(* IEC 61131-3 sources: volt/packages/volt-lsp-iec/test-corpus/lenze-mid/Device/Plc Logic/Application/Library Manager/SymbolicVarsBase, 107 files *)

(* ---- ADDRESSOFINTERFACEUNION.dut ---- *)
TYPE ADDRESSOFINTERFACEUNION :
UNION
	IITF : __SYSTEM.IQueryInterface;
	IBASETREENODE : IBaseTreeNode;
	PITF : POINTER TO BYTE;
END_UNION
END_TYPE

(* ---- BROWSEOPERATION.dut ---- *)
TYPE BROWSEOPERATION :
(
	FIND_CHILD := 0,
	BROWSE_DOWN,
	BROWSE_NEXT,
	BROWSE_UP
);
END_TYPE

(* ---- CALLGLUEFUNCTIONPARAMETERSET.dut ---- *)
TYPE CALLGLUEFUNCTIONPARAMETERSET :
STRUCT
	PARGUMENTBUFFER : POINTER TO BYTE;
	NARGUMENTBUFFERSIZE : __XWORD;
	ITYPEDESC : REFERENCE TO TypeDesc;
	PINSTANCE : POINTER TO BYTE;
	PINTERFACE : __SYSTEM.IQueryInterface;
	RESULT : RTS_IEC_RESULT;
END_STRUCT
END_TYPE

(* ---- DIRECTIOBITS16.dut ---- *)
TYPE DIRECTIOBITS16 :
STRUCT
	X0 : BIT;
	X1 : BIT;
	X2 : BIT;
	X3 : BIT;
	X4 : BIT;
	X5 : BIT;
	X6 : BIT;
	X7 : BIT;
	X8 : BIT;
	X9 : BIT;
	X10 : BIT;
	X11 : BIT;
	X12 : BIT;
	X13 : BIT;
	X14 : BIT;
	X15 : BIT;
END_STRUCT
END_TYPE

(* ---- DIRECTIOBITS8.dut ---- *)
TYPE DIRECTIOBITS8 :
STRUCT
	X0 : BIT;
	X1 : BIT;
	X2 : BIT;
	X3 : BIT;
	X4 : BIT;
	X5 : BIT;
	X6 : BIT;
	X7 : BIT;
END_STRUCT
END_TYPE

(* ---- GETTYPENODEOPTIONS.dut ---- *)
TYPE GETTYPENODEOPTIONS :
(
	NOOPTION := 0,
	GETBASETYPE := 16#1,
	GETBROWSETYPE := 16#2
);
END_TYPE

(* ---- IECOPCUAMAPPING.dut ---- *)
TYPE IECOPCUAMAPPING :
STRUCT
	IECTYPE : TypeClass;
	UATYPE : OpcUa_BuiltInType;
	CONVERSIONNEEDED : BOOL;
END_STRUCT
END_TYPE

(* ---- LOGGERSTRING.dut ---- *)
TYPE LOGGERSTRING : STRING(255);
END_TYPE

(* ---- NESTINGPATHENTRY.dut ---- *)
TYPE NESTINGPATHENTRY :
STRUCT
	PPROPERTYINFO : POINTER TO PropertyInfo;
	PREFERENCEINFO : POINTER TO BYTE;
	CONTAININGNODE : ILeafTreeNode;
	NNEXTOFFSET : __XWORD;
	PTYPENODE : REFERENCE TO TypeDesc;
END_STRUCT
END_TYPE

(* ---- NESTINGPATHINFORMATION.dut ---- *)
TYPE NESTINGPATHINFORMATION :
STRUCT
	NMAXDEPTH : UDINT;
	NELEMENTSUSED : UDINT;
	APATHINFO : ARRAY [0..5] OF NestingPathEntry;
END_STRUCT
END_TYPE

(* ---- NODEFLAGS.dut ---- *)
TYPE NODEFLAGS :
(
	LTNF_NONE := 16#0,
	LTNF_VAR := 16#1,
	LTNF_VAR_INPUT := 16#2,
	LTNF_VAR_OUTPUT := 16#4,
	LTNF_VAR_IN_OUT := 16#8,
	LTNF_VAR_EXEC := 16#10,
	LTNF_VAR_PROP := 16#20,
	LTNF_CALL_PROP := 16#40,
	LTNF_INHERITED_MEMBER := 16#10000
);
END_TYPE

(* ---- OPCUAMETADATATYPE.dut ---- *)
TYPE OPCUAMETADATATYPE :
(
	WELLKNOWNDATATYPEMETA := 0,
	OWNDATATYPEMETA,
	METHODMETA
);
END_TYPE

(* ---- OPCUAMETHODMETADATA.dut ---- *)
TYPE OPCUAMETHODMETADATA :
STRUCT
	INPUTARGUMENTS : OpcUa_NodeId;
	OUTPUTARGUMENTS : OpcUa_NodeId;
END_STRUCT
END_TYPE

(* ---- OPCUANODEMETADATA.dut ---- *)
TYPE OPCUANODEMETADATA :
STRUCT
	BROWSENAME : OpcUa_QualifiedName;
	DISPLAYNAME : OpcUa_LocalizedText;
	NODECLASS : OpcUa_NodeClass;
	DESCRIPTION : OpcUa_LocalizedText;
	EVENTNOTIFIER : OpcUa_Byte;
	REFERENCEPARENT : OpcUa_NodeId;
	TYPEDEFINITION : OpcUa_NodeId;
	ENTRYPOINT : OpcUa_NodeId;
END_STRUCT
END_TYPE

(* ---- OPCUAOWNDATATYPEMETADATA.dut ---- *)
TYPE OPCUAOWNDATATYPEMETADATA :
STRUCT
	PARENTID : OpcUa_NodeId;
	PARTENTREFERENCETYPE : OpcUa_NodeId;
END_STRUCT
END_TYPE

(* ---- OPCUATYPEMETADATA.dut ---- *)
TYPE OPCUATYPEMETADATA :
STRUCT
	METATYPE : OpcUaMetaDataType;
	DATA : OpcUaTypeMetaDataUnion;
END_STRUCT
END_TYPE

(* ---- OPCUATYPEMETADATAUNION.dut ---- *)
TYPE OPCUATYPEMETADATAUNION :
UNION
	WELLKNOWN : OpcUaWellKnownDataTypeMetaData;
	OWNDATATYPE : OpcUaOwnDataTypeMetaData;
	METHODDATA : OpcUaMethodMetaData;
END_UNION
END_TYPE

(* ---- OPCUAWELLKNOWNDATATYPEMETADATA.dut ---- *)
TYPE OPCUAWELLKNOWNDATATYPEMETADATA :
STRUCT
	NODEID : OpcUa_NodeId;
	ENCODINGID : OpcUa_NodeId;
END_STRUCT
END_TYPE

(* ---- PROPERTYINFO.dut ---- *)
TYPE PROPERTYINFO :
STRUCT
	PINSTANCE : POINTER TO BYTE;
	PPFGET : POINTER TO POINTER TO BYTE;
	PPFSET : POINTER TO POINTER TO BYTE;
	_NPROPOFFSETGET : INT;
	_NPROPOFFSETSET : INT;
END_STRUCT
END_TYPE

(* ---- PROPERTYINFOREMOTE.dut ---- *)
TYPE PROPERTYINFOREMOTE :
STRUCT
	AREACODE : INT;
	OFFSETGET : DINT;
	OFFSETSET : DINT;
END_STRUCT
END_TYPE

(* ---- SYMBOLICVARSBASEHANDLECONVERTER.dut ---- *)
TYPE SYMBOLICVARSBASEHANDLECONVERTER :
UNION
	HHANDLE : RTS_IEC_HANDLE;
	PBASENODE : IBaseTreeNode;
	PTYPEDESC : ITypeDesc;
END_UNION
END_TYPE

(* ---- GVL_LIBRARYDEFINES.gvl ---- *)
VAR_GLOBAL
	IECVARACCESS_VERSION_GE_3_1_3_0 : INT := 1;
	IECVARACCESS_VERSION_GE_3_2_0_1 : INT := 2;
	CMPID_IECVARACCESS : DWORD := 16#1007;
	IECVARACCESS_LIB_VERSION : DWORD := 16#3050340;
	CMPNAME_IECVARACCESS : STRING := 'IecVarAccess';
END_VAR

(* ---- IECUAMAPPING.gvl ---- *)
VAR_GLOBAL
	MAPPING : ARRAY [0..49] OF IecOpcUaMapping := [STRUCT(iecType := TYPE_BOOL, uaType := OpcUaType_Boolean), STRUCT(iecType := TYPE_BIT, uaType := OpcUaType_Boolean), STRUCT(iecType := TYPE_BYTE, uaType := OpcUaType_Byte), STRUCT(iecType := TYPE_WORD, uaType := OpcUaType_UInt16), STRUCT(iecType := TYPE_DWORD, uaType := OpcUaType_UInt32), STRUCT(iecType := TYPE_LWORD, uaType := OpcUaType_UInt64), STRUCT(iecType := TYPE_SINT, uaType := OpcUaType_SByte), STRUCT(iecType := TYPE_INT, uaType := OpcUaType_Int16), STRUCT(iecType := TYPE_DINT, uaType := OpcUaType_Int32), STRUCT(iecType := TYPE_LINT, uaType := OpcUaType_Int64), STRUCT(iecType := TYPE_USINT, uaType := OpcUaType_Byte), STRUCT(iecType := TYPE_UINT, uaType := OpcUaType_UInt16), STRUCT(iecType := TYPE_UDINT, uaType := OpcUaType_UInt32), STRUCT(iecType := TYPE_ULINT, uaType := OpcUaType_UInt64), STRUCT(iecType := TYPE_REAL, uaType := OpcUaType_Float), STRUCT(iecType := TYPE_LREAL, uaType := OpcUaType_Double), STRUCT(iecType := TYPE_STRING, uaType := OpcUaType_String), STRUCT(iecType := TYPE_WSTRING, uaType := OpcUaType_String), STRUCT(iecType := TYPE_TIME, uaType := OpcUaType_Int64), STRUCT(iecType := TYPE_DATE, uaType := OpcUaType_DateTime), STRUCT(iecType := TYPE_DATEANDTIME, uaType := OpcUaType_DateTime), STRUCT(iecType := TYPE_TIMEOFDAY, uaType := OpcUaType_UInt32), STRUCT(iecType := TYPE_POINTER, uaType := OpcUaType_Null), STRUCT(iecType := TYPE_REFERENCE, uaType := OpcUaType_Null), STRUCT(iecType := TYPE_SUBRANGE, uaType := OpcUaType_Null), STRUCT(iecType := TYPE_ENUM, uaType := OpcUaType_Null), STRUCT(iecType := TYPE_ARRAY, uaType := OpcUaType_Null), STRUCT(iecType := TYPE_PARAMS, uaType := OpcUaType_Null), STRUCT(iecType := TYPE_USERDEF, uaType := OpcUaType_ExtensionObject), STRUCT(iecType := TYPE_NONE, uaType := OpcUaType_Null), STRUCT(iecType := TYPE_ANY, uaType := OpcUaType_Null), STRUCT(iecType := TYPE_ANYBIT, uaType := OpcUaType_Null), STRUCT(iecType := TYPE_ANYDATE, uaType := OpcUaType_Null), STRUCT(iecType := TYPE_ANYINT, uaType := OpcUaType_Null), STRUCT(iecType := TYPE_ANYNUM, uaType := OpcUaType_Null), STRUCT(iecType := TYPE_ANYREAL, uaType := OpcUaType_Null), STRUCT(iecType := TYPE_LAZY, uaType := OpcUaType_Null), STRUCT(iecType := TYPE_LTIME, uaType := OpcUaType_Int64), STRUCT(iecType := TYPE_BITCONST, uaType := OpcUaType_Null), STRUCT(iecType := TYPE_UXINT, uaType := OpcUaType_Null), STRUCT(iecType := TYPE_XWORD, uaType := OpcUaType_Null), STRUCT(iecType := TYPE_XINT, uaType := OpcUaType_Null), STRUCT(iecType := TYPE_XSRTING, uaType := OpcUaType_Null), STRUCT(iecType := TYPE_VARLENARRAY, uaType := OpcUaType_Null), STRUCT(iecType := TYPE_ANYSTRING, uaType := OpcUaType_Null), STRUCT(iecType := TYPE_VECTOR, uaType := OpcUaType_Null), STRUCT(iecType := TYPE_LDATE, uaType := OpcUaType_Null), STRUCT(iecType := TYPE_LDATEANDTIME, uaType := OpcUaType_Null), STRUCT(iecType := TYPE_LTIMEOFDAY, uaType := OpcUaType_Null), STRUCT(iecType := TYPE_INTERFACE, uaType := OpcUaType_Null)];
	SECS_BETWEEN_EPOCHS : LINT := 11644473600;
	SECS_TO_100NS : LINT := 10000000;
END_VAR

(* ---- INTERFACEIDS.gvl ---- *)
VAR_GLOBAL
	ITFID_ICOLLECTSSECONDOFFSET : DWORD := 16#1003;
	ITFID_ICOLLECTSPROPERTYINFORMATION : DWORD := 16#1004;
	ITFID_ILEAFTREENODE : DWORD := 16#1006;
	ITFID_IBRANCHTREENODE : DWORD := 16#1011;
	ITFID_IMEMBERINDEX : DWORD := 16#1012;
	ITFID_IARRAYNOTIFIABLE : DWORD := 16#1030;
	ITFID_IVARIABLEINFORMATIONCOMBINED : DWORD := 16#1105;
	ITFID_ITREEWALKER : DWORD := 16#1111;
END_VAR

(* ---- POUTYPECLASS.gvl ---- *)
VAR_GLOBAL
	TYPE_POU_FUNCTION : INT := 16#100;
	TYPE_POU_FUNCTION_BLOCK : INT := 16#200;
	TYPE_POU_PROGRAM : INT := 16#300;
	TYPE_POU_STRUCTURE : INT := 16#400;
	TYPE_POU_UNION : INT := 16#500;
	TYPE_POU_UABUILTIN : INT := 16#1000;
END_VAR

(* ---- TYPECLASSFLAGBITS.gvl ---- *)
VAR_GLOBAL
	TYPECLASS_FLAG_ALIAS : INT := 16#900;
	TYPECLASS_MAGIC_PROPERTY : INT := ANY_TO_INT(16#E000);
	TYPECLASS_BITMASK_TYPECLASS : INT := 16#FF;
	TYPECLASS_BITMASK_POUTYPE : INT := 16#700;
	TYPECLASS_BITMASK_FLAGS : INT := ANY_TO_INT(16#F800);
END_VAR

(* ---- TYPEFLAGS.gvl ---- *)
VAR_GLOBAL
	TYPEFLAG_REFERENCE : DWORD := 16#1;
END_VAR

(* ---- IARRAYNOTIFIABLE.itf ---- *)
INTERFACE IARRAYNOTIFIABLE
END_INTERFACE

METHOD ARRAYACCESSDETECTED
VAR_INPUT
	PSTR : POINTER TO STRING;
	LENGTH : INT;
END_VAR
END_METHOD

(* ---- IBRANCHTREENODE.itf ---- *)
INTERFACE IBRANCHTREENODE
END_INTERFACE

METHOD GETATTRIBUTEBYINDEX : POINTER TO STRING
VAR_INPUT
	WINDEX : WORD;
END_VAR
END_METHOD

METHOD GETNAMESPACENODEFLAGS : IecVarAccess_Interfaces.NamespaceNodeFlags
VAR_INPUT
	PRESULT : POINTER TO UDINT;
END_VAR
END_METHOD

METHOD GETNUMOFATTRIBUTES : WORD
END_METHOD

(* ---- ILEAFTREENODE.itf ---- *)
INTERFACE ILEAFTREENODE
END_INTERFACE

METHOD EXECUTECALL : RTS_IEC_RESULT
VAR_INPUT
	VARINFO : REFERENCE TO VariableInformation;
	PARGUMENTBUFFER : POINTER TO BYTE;
	NARGUMENTBUFFERSIZE : __XWORD;
	CALLEXECUTORFUNCTION : POINTER TO POINTER TO BYTE;
	EXECUTABLETYPEDESC : REFERENCE TO TypeDesc;
END_VAR
END_METHOD

METHOD EXECUTECALL2 : RTS_IEC_RESULT
VAR_INPUT
	VARINFO : REFERENCE TO VariableInformation;
	PARGUMENTBUFFER : POINTER TO BYTE;
	NARGUMENTBUFFERSIZE : __XWORD;
END_VAR
END_METHOD

METHOD GET : __XWORD
VAR_INPUT
	PDEST : POINTER TO BYTE;
	VARINFO : REFERENCE TO VariableInformation;
	DWSIZE : __XWORD;
	PRESULT : POINTER TO RTS_IEC_RESULT;
END_VAR
END_METHOD

METHOD GETACCESSRIGHTS : BYTE
END_METHOD

METHOD GETACCESSRIGHTS2 : BYTE
VAR_INPUT
	VARINFO : REFERENCE TO VariableInformation;
	BGETUSERRIGHTS : BOOL;
END_VAR
END_METHOD

METHOD GETADDRESS : POINTER TO BYTE
END_METHOD

METHOD GETADDRESS3 : POINTER TO BYTE
VAR_INPUT
	PVARIABLEINFORMATION : POINTER TO VariableInformationStruct;
END_VAR
END_METHOD

METHOD GETATTRIBUTEBYINDEX : POINTER TO STRING
VAR_INPUT
	WINDEX : WORD;
END_VAR
END_METHOD

METHOD GETCLIENTOFFSET : DWORD
END_METHOD

METHOD GETFLAGS : NodeFlags
END_METHOD

METHOD GETNAMESPACENODEFLAGS : IecVarAccess_Interfaces.NamespaceNodeFlags
VAR_INPUT
	PRESULT : POINTER TO UDINT;
END_VAR
END_METHOD

METHOD GETNUMOFATTRIBUTES : WORD
END_METHOD

METHOD GETSIZE : __XWORD
VAR_INPUT
	VARINFO : REFERENCE TO VariableInformation;
	PRESULT : POINTER TO RTS_IEC_RESULT;
END_VAR
END_METHOD

METHOD GETTYPE : REFERENCE TO TypeDesc
VAR_INPUT
	VARINFO : REFERENCE TO VariableInformation;
	OPTIONS : WORD;
END_VAR
END_METHOD

METHOD NODEFOUND : UDINT
VAR_INPUT
	VARINFO : REFERENCE TO VariableInformation;
	BDIRECTCHILDFOUND : BOOL;
END_VAR
END_METHOD

METHOD SET : __XWORD
VAR_INPUT
	PSRC : POINTER TO BYTE;
	VARINFO : REFERENCE TO VariableInformation;
	DWSIZE : __XWORD;
	PRESULT : POINTER TO RTS_IEC_RESULT;
END_VAR
END_METHOD

METHOD SWAP2 : __XWORD
VAR_INPUT
	PDATA : POINTER TO BYTE;
	VARINFO : REFERENCE TO VariableInformation;
	BMOTOROLA : BOOL;
	PRESULT : POINTER TO RTS_IEC_RESULT;
END_VAR
END_METHOD

(* ---- IMEMBERINDEX.itf ---- *)
INTERFACE IMEMBERINDEX
END_INTERFACE

(* ---- IOPCUADATATYPEFINDCHILDBYBROWSENAME.itf ---- *)
INTERFACE IOPCUADATATYPEFINDCHILDBYBROWSENAME
END_INTERFACE

METHOD GETFIRSTCHILDBYBROWSENAME : ITreeWalker
VAR_INPUT
	PBROWSENAME : POINTER TO OpcUa_QualifiedName;
	VARINFO : REFERENCE TO VariableInformation;
END_VAR
VAR_OUTPUT
	RESULT : RTS_IEC_RESULT;
END_VAR
END_METHOD

(* ---- IOPCUADATATYPEMETADATA.itf ---- *)
INTERFACE IOPCUADATATYPEMETADATA
END_INTERFACE

METHOD GETDATATYPEID : RTS_IEC_RESULT
VAR_OUTPUT
	PDATATYPEID : POINTER TO OpcUa_NodeId;
END_VAR
END_METHOD

METHOD GETENCODINGNODEID : RTS_IEC_RESULT
VAR_OUTPUT
	PENCODINGID : POINTER TO OpcUa_NodeId;
END_VAR
END_METHOD

METHOD GETMETHODARGUMENTS : RTS_IEC_RESULT
VAR_OUTPUT
	PINPUTARGUMENTS : POINTER TO OpcUa_NodeId;
	POUTPUTARGUMENTS : POINTER TO OpcUa_NodeId;
END_VAR
END_METHOD

METHOD GETPARENTNODE : RTS_IEC_RESULT
VAR_OUTPUT
	PPARENTNODE : POINTER TO OpcUa_NodeId;
END_VAR
END_METHOD

METHOD GETPARENTREFERENCETYPE : RTS_IEC_RESULT
VAR_OUTPUT
	PPARENTREFERENCETYPE : POINTER TO OpcUa_NodeId;
END_VAR
END_METHOD

METHOD ISWELLKNOWNTYPE : BOOL
END_METHOD

(* ---- IOPCUAINSTANCEMETADATA.itf ---- *)
INTERFACE IOPCUAINSTANCEMETADATA
END_INTERFACE

METHOD GETBROWSENAME : RTS_IEC_RESULT
VAR_OUTPUT
	PBROWSENAME : POINTER TO OpcUa_QualifiedName;
END_VAR
END_METHOD

METHOD GETDESCRIPTION : RTS_IEC_RESULT
VAR_OUTPUT
	PDESCRIPTION : POINTER TO OpcUa_LocalizedText;
END_VAR
END_METHOD

METHOD GETDISPLAYNAME : RTS_IEC_RESULT
VAR_OUTPUT
	PDISPLAYNAME : POINTER TO OpcUa_LocalizedText;
END_VAR
END_METHOD

METHOD GETENTRYPOINT : RTS_IEC_RESULT
VAR_OUTPUT
	ISENTRYPOINT : BOOL;
	PENTRYPOINT : POINTER TO CmpOPCUAStack_Interfaces.OpcUa_NodeId;
END_VAR
END_METHOD

METHOD GETEVENTNOTIFIER : RTS_IEC_RESULT
VAR_OUTPUT
	EVENTNOTIFIER : OpcUa_Byte;
END_VAR
END_METHOD

METHOD GETNODECLASS : RTS_IEC_RESULT
VAR_OUTPUT
	NODECLASS : OpcUa_NodeClass;
END_VAR
END_METHOD

METHOD GETPARENTREFERENCETYPE : RTS_IEC_RESULT
VAR_OUTPUT
	PREFERENCETYPE : POINTER TO OpcUa_NodeId;
END_VAR
END_METHOD

METHOD GETTYPEDEFINITION : RTS_IEC_RESULT
VAR_OUTPUT
	PTYPEDEFINITION : POINTER TO OpcUa_NodeId;
END_VAR
END_METHOD

(* ---- ISEARCHCALLBACKS.itf ---- *)
INTERFACE ISEARCHCALLBACKS
END_INTERFACE

METHOD IGNOREROOTNODE : BOOL
VAR_INPUT
	PNODE : ITreeWalker;
	VARINFO : REFERENCE TO VariableInformation;
END_VAR
END_METHOD

METHOD NODEFOUND
VAR_INPUT
	PNODE : ITreeWalker;
	VARINFO : REFERENCE TO VariableInformation;
	XROOTNODE : BOOL;
END_VAR
END_METHOD

METHOD NODENOTFOUND : ITreeWalker
VAR_INPUT
	PPARENT : ITreeWalker;
	SZCHILDNAME : POINTER TO BYTE;
	NAMELEN : __XWORD;
	SYMBOLSSETS : DWORD;
	VARINFO : REFERENCE TO VariableInformation;
	XROOTNODE : BOOL;
END_VAR
VAR_IN_OUT
	CONSUMED : __XWORD;
END_VAR
END_METHOD

(* ---- ITREEWALKER.itf ---- *)
INTERFACE ITREEWALKER
END_INTERFACE

METHOD ASBASETREENODE : IBaseTreeNode
END_METHOD

METHOD FINDCHILD : ITreeWalker
VAR_INPUT
	SZCHILDNAME : POINTER TO BYTE;
	NAMELEN : __XWORD;
	SYMBOLSSETS : DWORD;
	VARINFO : REFERENCE TO VariableInformation;
	PRESULT : POINTER TO RTS_IEC_RESULT;
END_VAR
VAR_IN_OUT
	TYPESYSTEMREACHED : BOOL;
END_VAR
END_METHOD

METHOD GETCHILDBYINDEX : ITreeWalker
VAR_INPUT
	IINDEX : DINT;
	USERACCESSRIGHTS : BYTE;
	SYMBOLSSETS : DWORD;
END_VAR
VAR_OUTPUT
	XOUTOFRANGE : BOOL;
END_VAR
END_METHOD

METHOD GETFIRSTCHILD : ITreeWalker
VAR_INPUT
	USERACCESSRIGHTS : BYTE;
	SYMBOLSSETS : DWORD;
END_VAR
END_METHOD

METHOD GETFULLPATH : DINT
VAR_INPUT
	PBUFFER : POINTER TO STRING;
	DIBUFFERSIZE : DINT;
END_VAR
VAR_OUTPUT
	BROOT_NODE : BOOL;
	BEMPTYNAMESPACENODE : BOOL;
END_VAR
END_METHOD

METHOD GETPARENT : ITreeWalker
VAR_INPUT
	USERACCESSRIGHTS : BYTE;
	SYMBOLSSETS : DWORD;
END_VAR
END_METHOD

METHOD GETSIBLING : ITreeWalker
VAR_INPUT
	USERACCESSRIGHTS : BYTE;
	SYMBOLSSETS : DWORD;
END_VAR
END_METHOD

METHOD ISVISIBLE : BOOL
VAR_INPUT
	USERACCESSRIGHTS : BYTE;
	SYMBOLSSETS : DWORD;
END_VAR
END_METHOD

METHOD GETCHILDBYBROWSENAME : ITreeWalker
VAR_INPUT
	PBROWSENAME : POINTER TO OpcUa_QualifiedName;
	VARINFO : REFERENCE TO VariableInformation;
END_VAR
END_METHOD

METHOD GETNEXTBYBROWSENAME : ITreeWalker
VAR_INPUT
	PBROWSENAME : POINTER TO OpcUa_QualifiedName;
	VARINFO : REFERENCE TO VariableInformation;
END_VAR
END_METHOD

(* ---- ADDRESSOFIBASETREENODE.pou ---- *)
FUNCTION ADDRESSOFIBASETREENODE : POINTER TO BYTE
VAR_INPUT
	IBASETREENODE : IBaseTreeNode;
END_VAR
END_FUNCTION

(* ---- ADDRESSOFINTERFACE.pou ---- *)
FUNCTION ADDRESSOFINTERFACE : POINTER TO BYTE
VAR_INPUT
	IITF : __SYSTEM.IQueryInterface;
END_VAR
END_FUNCTION

(* ---- ASCIIUPPER.pou ---- *)
FUNCTION ASCIIUPPER : BYTE
VAR_INPUT
	CHARACTER : BYTE;
END_VAR
END_FUNCTION

(* ---- CALCULATEPROPERTYBUFFERSIZE.pou ---- *)
FUNCTION CALCULATEPROPERTYBUFFERSIZE : __XWORD
VAR_INPUT
	DATATYPE : REFERENCE TO TypeDesc;
END_VAR
END_FUNCTION

(* ---- CALLGLUEDESERIALIZEPARAMETERS.pou ---- *)
FUNCTION CALLGLUEDESERIALIZEPARAMETERS : RTS_IEC_RESULT
VAR_INPUT
	PARGUMENTBUFFER : POINTER TO BYTE;
	NARGUMENTBUFFERSIZE : __XWORD;
	ITYPEDESC : REFERENCE TO TypeDesc;
	PPARSEDARGUMENTS : POINTER TO BYTE;
	NPARSEDARGUMENTSIZE : __XWORD;
END_VAR
END_FUNCTION

(* ---- CALLGLUESERIALIZERETURNVALUES.pou ---- *)
FUNCTION CALLGLUESERIALIZERETURNVALUES : RTS_IEC_RESULT
VAR_INPUT
	PARGUMENTBUFFER : POINTER TO BYTE;
	NARGUMENTBUFFERSIZE : __XWORD;
	ITYPEDESC : REFERENCE TO TypeDesc;
	PPARSEDARGUMENTS : POINTER TO BYTE;
	NPARSEDARGUMENTSIZE : __XWORD;
END_VAR
END_FUNCTION

(* ---- COMPAREBROWSENAME.pou ---- *)
FUNCTION COMPAREBROWSENAME : DINT
VAR_INPUT
	NAME1 : POINTER TO OpcUa_QualifiedName;
	NAME2 : POINTER TO OpcUa_QualifiedName;
END_VAR
END_FUNCTION

(* ---- CONVERTTOIBRANCHTREENODE.pou ---- *)
FUNCTION CONVERTTOIBRANCHTREENODE : IBranchTreeNode
VAR_INPUT
	PNODE : IBaseTreeNode;
END_VAR
END_FUNCTION

(* ---- CONVERTTOILEAFTREENODE.pou ---- *)
FUNCTION CONVERTTOILEAFTREENODE : ILeafTreeNode
VAR_INPUT
	PNODE : IBaseTreeNode;
END_VAR
END_FUNCTION

(* ---- CONVERTTOITREEWALKER.pou ---- *)
FUNCTION CONVERTTOITREEWALKER : ITreeWalker
VAR_INPUT
	PNODE : IBaseTreeNode;
END_VAR
END_FUNCTION

(* ---- FINDBYBROWSENAME.pou ---- *)
FUNCTION FINDBYBROWSENAME : POINTER TO SymbolsBaseNode
VAR_INPUT
	LIST : POINTER TO POINTER TO SymbolsBaseNode;
	NUMELEMENTS : DINT;
	PBROWSENAME : POINTER TO OpcUa_QualifiedName;
END_VAR
VAR_OUTPUT
	INDEX : DINT;
END_VAR
END_FUNCTION

(* ---- FINDNEXTBYBROWSENAME.pou ---- *)
FUNCTION FINDNEXTBYBROWSENAME : POINTER TO SymbolsBaseNode
VAR_INPUT
	LIST : POINTER TO POINTER TO SymbolsBaseNode;
	NUMELEMENTS : DINT;
	PBROWSENAME : POINTER TO OpcUa_QualifiedName;
	VARINFO : REFERENCE TO VariableInformation;
END_VAR
VAR_OUTPUT
	RESULT : RTS_IEC_RESULT;
END_VAR
VAR_IN_OUT
	INDEX : DINT;
END_VAR
END_FUNCTION

(* ---- HEXSTRING.pou ---- *)
FUNCTION HEXSTRING : STRING
VAR_INPUT
	UDIVALUE : __UXINT;
END_VAR
END_FUNCTION

(* ---- ISACCEPTEDLEAFNODE.pou ---- *)
FUNCTION ISACCEPTEDLEAFNODE : BOOL
VAR_INPUT
	NITYPE : INT;
END_VAR
END_FUNCTION

(* ---- ISINVALIDMEMORYADDRESS.pou ---- *)
FUNCTION ISINVALIDMEMORYADDRESS : BOOL
VAR_INPUT
	PDATA : POINTER TO BYTE;
	XWSIZE : __XWORD;
	BWRITE : BOOL;
	PRESULT : POINTER TO RTS_IEC_RESULT;
END_VAR
END_FUNCTION

(* ---- ITREEWALKER_TOSTRING.pou ---- *)
FUNCTION ITREEWALKER_TOSTRING : LoggerString
VAR_INPUT
	ITREEWALKER : ITreeWalker;
END_VAR
END_FUNCTION

(* ---- LEAFTREENODE_TOSTRING.pou ---- *)
FUNCTION LEAFTREENODE_TOSTRING : LoggerString
VAR_INPUT
	LEAFTREENODE : POINTER TO LeafTreeNode;
END_VAR
END_FUNCTION

(* ---- LOGERROR.pou ---- *)
FUNCTION LOGERROR
VAR_INPUT
	STR : LoggerString;
END_VAR
END_FUNCTION

(* ---- LOGINFO.pou ---- *)
FUNCTION LOGINFO
VAR_INPUT
	STR : LoggerString;
END_VAR
END_FUNCTION

(* ---- LOGSTRING.pou ---- *)
FUNCTION LOGSTRING
VAR_INPUT
	STR : LoggerString;
	LOGCLASS : UDINT := CmpLog.LogClass.LOG_INFO;
END_VAR
END_FUNCTION

(* ---- MEMCPY.pou ---- *)
FUNCTION MEMCPY : __XWORD
VAR_INPUT
	PBYDEST : POINTER TO BYTE;
	PBYSRC : POINTER TO BYTE;
	DWSIZE : __XWORD;
END_VAR
END_FUNCTION

(* ---- MEMSET.pou ---- *)
FUNCTION MEMSET : __XWORD
VAR_INPUT
	PBYDEST : POINTER TO BYTE;
	BYVALUE : BYTE;
	DWSIZE : __XWORD;
END_VAR
END_FUNCTION

(* ---- PSTRCAT.pou ---- *)
FUNCTION PSTRCAT : DINT
VAR_INPUT
	PSTDEST : POINTER TO STRING;
	PSTSRC : POINTER TO STRING;
	DIDESTSIZE : DINT;
END_VAR
END_FUNCTION

(* ---- PSTRCMP.pou ---- *)
FUNCTION PSTRCMP : INT
VAR_INPUT
	PSTR1 : POINTER TO STRING;
	PSTR2 : POINTER TO STRING;
END_VAR
END_FUNCTION

(* ---- PSTRICMP.pou ---- *)
FUNCTION PSTRICMP : INT
VAR_INPUT
	PSTR1 : POINTER TO STRING;
	PSTR2 : POINTER TO STRING;
END_VAR
END_FUNCTION

(* ---- PSTRLEN.pou ---- *)
FUNCTION PSTRLEN : DINT
VAR_INPUT
	PSTRING : POINTER TO STRING;
END_VAR
END_FUNCTION

(* ---- PSTRLENUNTIL.pou ---- *)
FUNCTION PSTRLENUNTIL : DINT
VAR_INPUT
	PST : POINTER TO STRING;
	STTOKENDELIMITERS : STRING;
END_VAR
END_FUNCTION

(* ---- PSTRNICMP.pou ---- *)
FUNCTION PSTRNICMP : INT
VAR_INPUT
	PSTR1 : POINTER TO STRING;
	PSTR2 : POINTER TO STRING;
	N : __XWORD;
END_VAR
END_FUNCTION

(* ---- REPARSEIOMEMORYACCESSEXPRESSION.pou ---- *)
FUNCTION REPARSEIOMEMORYACCESSEXPRESSION : BOOL
VAR_INPUT
	STDESTINATION : REFERENCE TO STRING(255);
	PSZSOURCE : POINTER TO STRING(255);
END_VAR
END_FUNCTION

(* ---- RTSBROWSEINFO_TOSTRING.pou ---- *)
FUNCTION RTSBROWSEINFO_TOSTRING : LoggerString
VAR_INPUT
	PBROWSEINFO : POINTER TO RtsBrowseInfo;
END_VAR
END_FUNCTION

(* ---- SETRESULT.pou ---- *)
FUNCTION SETRESULT
VAR_INPUT
	PRESULT : POINTER TO RTS_IEC_RESULT;
	RESULT : RTS_IEC_RESULT;
END_VAR
END_FUNCTION

(* ---- STRINGPOINTER_TOSTRING.pou ---- *)
FUNCTION STRINGPOINTER_TOSTRING : LoggerString
VAR_INPUT
	PSTRING : POINTER TO STRING;
END_VAR
END_FUNCTION

(* ---- TYPEDESC_TOSTRING.pou ---- *)
FUNCTION TYPEDESC_TOSTRING : LoggerString
VAR_INPUT
	TYPEDESC : REFERENCE TO TypeDesc;
END_VAR
END_FUNCTION

(* ---- TYPEHASCOMPLETEBLITTABLELAYOUT.pou ---- *)
FUNCTION TYPEHASCOMPLETEBLITTABLELAYOUT : BOOL
VAR_INPUT
	TYPEDESC : REFERENCE TO TypeDesc;
END_VAR
END_FUNCTION

(* ---- BRANCHTREENODE.pou ---- *)
FUNCTION_BLOCK BRANCHTREENODE EXTENDS SymbolsBranchNode
VAR
	_IBRANCHTREENODE : IBranchTreeNode;
	_BNODEVALID : BOOL;
	ABSTRNODETYPE : INT;
END_VAR
END_FUNCTION_BLOCK

METHOD GETATTRIBUTEBYINDEX : POINTER TO STRING
VAR_INPUT
	WINDEX : WORD;
END_VAR
END_METHOD

METHOD GETNAMESPACENODEFLAGS : IecVarAccess_Interfaces.NamespaceNodeFlags
VAR_INPUT
	PRESULT : POINTER TO UDINT;
END_VAR
END_METHOD

METHOD GETNUMOFATTRIBUTES : WORD
END_METHOD

METHOD FB_EXIT : BOOL
VAR_INPUT
	BINCOPYCODE : BOOL;
END_VAR
END_METHOD

METHOD FB_INIT : BOOL
VAR_INPUT
	BINITRETAINS : BOOL;
	BINCOPYCODE : BOOL;
END_VAR
END_METHOD

METHOD QUERYINTERFACE : POINTER TO POINTER TO BYTE
VAR_INPUT
	IID : DWORD;
	PRESULT : POINTER TO UDINT;
END_VAR
END_METHOD

(* ---- BRANCHTREENODEOPCUA.pou ---- *)
FUNCTION_BLOCK BRANCHTREENODEOPCUA EXTENDS BranchTreeNode
VAR
	_NUMOFATTRIBUTES : WORD;
	_PATTRIBUTES : POINTER TO ARRAY [0..0] OF POINTER TO STRING;
	_ENAMESPACENODEFLAGS : IecVarAccess_Interfaces.NamespaceNodeFlags;
END_VAR
END_FUNCTION_BLOCK

METHOD GETATTRIBUTEBYINDEX : POINTER TO STRING
VAR_INPUT
	WINDEX : WORD;
END_VAR
END_METHOD

METHOD GETNAMESPACENODEFLAGS : IecVarAccess_Interfaces.NamespaceNodeFlags
VAR_INPUT
	PRESULT : POINTER TO UDINT;
END_VAR
END_METHOD

METHOD GETNUMOFATTRIBUTES : WORD
END_METHOD

(* ---- LEAFTREENODE.pou ---- *)
FUNCTION_BLOCK LEAFTREENODE EXTENDS SymbolsBaseNode
VAR
	_ITYPEDESC : REFERENCE TO TypeDesc;
	_ILEAFTREENODE : ILeafTreeNode;
	_PADDRESS : POINTER TO BYTE;
	_ACCESSRIGHTS : BYTE;
	_DWREADMASK : DWORD := ANY_TO_DWORD(-1);
	_DWWRITEMASK : DWORD := ANY_TO_DWORD(-1);
	_DWEXECUTEMASK : DWORD := ANY_TO_DWORD(-1);
	_BNODEVALID : BOOL;
	ABSTRNODETYPE : INT;
	ISSTATICVARWITHINNONSTATICFBINSTANCE : BOOL;
	NAME : POINTER TO STRING;
END_VAR
END_FUNCTION_BLOCK

METHOD CHECKPROPERTYANDREFERENCE : RTS_IEC_RESULT
VAR_INPUT
	VARINFO : REFERENCE TO VariableInformation;
END_VAR
VAR_OUTPUT
	ISPROPERTY : BOOL;
	ISREFERENCE : BOOL;
END_VAR
END_METHOD

METHOD COMPARENAME : INT
VAR_INPUT
	PSTNAME : POINTER TO BYTE;
	NAMELEN : __XWORD;
END_VAR
END_METHOD

METHOD CONVERTTOITREENODE : ITreeWalker
VAR_INPUT
	PNODE : IInstancePathBuildingNode;
END_VAR
END_METHOD

METHOD EXECUTECALL : RTS_IEC_RESULT
VAR_INPUT
	VARINFO : REFERENCE TO VariableInformation;
	PARGUMENTBUFFER : POINTER TO BYTE;
	NARGUMENTBUFFERSIZE : __XWORD;
	CALLEXECUTORFUNCTION : POINTER TO POINTER TO BYTE;
	EXECUTABLETYPEDESC : REFERENCE TO TypeDesc;
END_VAR
END_METHOD

METHOD EXECUTECALL2 : SysTypes.RTS_IEC_RESULT
VAR_INPUT
	VARINFO : REFERENCE TO VariableInformation;
	PARGUMENTBUFFER : POINTER TO BYTE;
	NARGUMENTBUFFERSIZE : __XWORD;
END_VAR
END_METHOD

METHOD FINDCHILD : ITreeWalker
VAR_INPUT
	SZCHILDNAME : POINTER TO BYTE;
	NAMELEN : __XWORD;
	SYMBOLSSETS : DWORD;
	VARINFO : REFERENCE TO VariableInformation;
	PRESULT : POINTER TO RTS_IEC_RESULT;
END_VAR
VAR_IN_OUT
	TYPESYSTEMREACHED : BOOL;
END_VAR
END_METHOD

METHOD GETACCESSRIGHTS : BYTE
END_METHOD

METHOD GETACCESSRIGHTS2 : BYTE
VAR_INPUT
	VARINFO : REFERENCE TO VariableInformation;
	BGETUSERRIGHTS : BOOL;
END_VAR
END_METHOD

METHOD GETADDRESS : POINTER TO BYTE
END_METHOD

METHOD GETADDRESS3 : POINTER TO BYTE
VAR_INPUT
	PVARIABLEINFORMATION : POINTER TO VariableInformationStruct;
END_VAR
END_METHOD

METHOD GETATTRIBUTEBYINDEX : POINTER TO STRING
VAR_INPUT
	WINDEX : WORD;
END_VAR
END_METHOD

METHOD GETCHILDBYBROWSENAME : ITreeWalker
VAR_INPUT
	PBROWSENAME : POINTER TO OpcUa_QualifiedName;
	VARINFO : REFERENCE TO VariableInformation;
END_VAR
END_METHOD

METHOD GETCLIENTOFFSET : DWORD
END_METHOD

METHOD GETFLAGS : NodeFlags
END_METHOD

METHOD GETNAMESPACENODEFLAGS : IecVarAccess_Interfaces.NamespaceNodeFlags
VAR_INPUT
	PRESULT : POINTER TO UDINT;
END_VAR
END_METHOD

METHOD GETNUMOFATTRIBUTES : WORD
END_METHOD

METHOD GETSIZE : __XWORD
VAR_INPUT
	VARINFO : REFERENCE TO VariableInformation;
	PRESULT : POINTER TO RTS_IEC_RESULT;
END_VAR
END_METHOD

METHOD GETSTATICVARLEAFTREENODEADDR : POINTER TO LeafTreeNode
END_METHOD

METHOD GETSTATICVARSYMBOLSBASENODEADDR : POINTER TO SymbolsBaseNode
END_METHOD

METHOD GETTYPE : REFERENCE TO TypeDesc
VAR_INPUT
	VARINFO : REFERENCE TO VariableInformation;
	OPTIONS : WORD;
END_VAR
END_METHOD

METHOD GET : __XWORD
VAR_INPUT
	PDEST : POINTER TO BYTE;
	VARINFO : REFERENCE TO VariableInformation;
	DWSIZE : __XWORD;
	PRESULT : POINTER TO RTS_IEC_RESULT;
END_VAR
END_METHOD

METHOD NODEFOUND : UDINT
VAR_INPUT
	VARINFO : REFERENCE TO VariableInformation;
	BDIRECTCHILDFOUND : BOOL;
END_VAR
END_METHOD

METHOD RESOLVESTATICVAR : ITreeWalker
END_METHOD

METHOD SET : __XWORD
VAR_INPUT
	PSRC : POINTER TO BYTE;
	VARINFO : REFERENCE TO VariableInformation;
	DWSIZE : __XWORD;
	PRESULT : POINTER TO RTS_IEC_RESULT;
END_VAR
END_METHOD

METHOD SWAP2 : __XWORD
VAR_INPUT
	PDATA : POINTER TO BYTE;
	VARINFO : REFERENCE TO VariableInformation;
	BMOTOROLA : BOOL;
	PRESULT : POINTER TO RTS_IEC_RESULT;
END_VAR
END_METHOD

METHOD FB_EXIT : BOOL
VAR_INPUT
	BINCOPYCODE : BOOL;
END_VAR
END_METHOD

METHOD FB_INIT : BOOL
VAR_INPUT
	BINITRETAINS : BOOL;
	BINCOPYCODE : BOOL;
END_VAR
END_METHOD

METHOD QUERYINTERFACE : POINTER TO POINTER TO BYTE
VAR_INPUT
	IID : DWORD;
	PRESULT : POINTER TO UDINT;
END_VAR
END_METHOD

(* ---- LEAFTREENODEOPCUA.pou ---- *)
FUNCTION_BLOCK LEAFTREENODEOPCUA EXTENDS LeafTreeNode
VAR
	_NUMOFATTRIBUTES : WORD;
	_PATTRIBUTES : POINTER TO ARRAY [0..0] OF POINTER TO STRING;
	_ENAMESPACENODEFLAGS : IecVarAccess_Interfaces.NamespaceNodeFlags;
END_VAR
END_FUNCTION_BLOCK

METHOD GETATTRIBUTEBYINDEX : POINTER TO STRING
VAR_INPUT
	WINDEX : WORD;
END_VAR
END_METHOD

METHOD GETNAMESPACENODEFLAGS : IecVarAccess_Interfaces.NamespaceNodeFlags
VAR_INPUT
	PRESULT : POINTER TO UDINT;
END_VAR
END_METHOD

METHOD GETNUMOFATTRIBUTES : WORD
END_METHOD

(* ---- LEAFTREENODETYPEMEMBER.pou ---- *)
FUNCTION_BLOCK LEAFTREENODETYPEMEMBER EXTENDS LeafTreeNode
VAR
	_CLIENTOFFSET : DWORD;
END_VAR
END_FUNCTION_BLOCK

METHOD GETCLIENTOFFSET : DWORD
END_METHOD

METHOD GETNEXTBYBROWSENAME : ITreeWalker
VAR_INPUT
	PBROWSENAME : POINTER TO OpcUa_QualifiedName;
	VARINFO : REFERENCE TO VariableInformation;
END_VAR
END_METHOD

(* ---- LEAFTREENODETYPEMEMBEROPCUA.pou ---- *)
FUNCTION_BLOCK LEAFTREENODETYPEMEMBEROPCUA EXTENDS LeafTreeNodeTypeMember
VAR
	_DWFLAGS : NodeFlags;
	_NUMOFATTRIBUTES : WORD;
	_PATTRIBUTES : POINTER TO ARRAY [0..0] OF POINTER TO STRING;
END_VAR
END_FUNCTION_BLOCK

METHOD GETATTRIBUTEBYINDEX : POINTER TO STRING
VAR_INPUT
	WINDEX : WORD;
END_VAR
END_METHOD

METHOD GETFLAGS : NodeFlags
END_METHOD

METHOD GETNUMOFATTRIBUTES : WORD
END_METHOD

(* ---- SYMBOLICVARNODEACCESSOR.pou ---- *)
FUNCTION_BLOCK SYMBOLICVARNODEACCESSOR
VAR
	_UDISYMBOLCONFIGCRC : UDINT;
	_ACCESSMASK : __XWORD;
	_TYPELIST : POINTER TO ARRAY [0..0] OF POINTER TO TypeDesc;
	_NUMOFTYPES : DINT;
	_BSYMBOLSVALID : BOOL;
	_CALLEXECUTORFUNCTION : POINTER TO POINTER TO BYTE;
	_METHODCALLTYPEDESCS : POINTER TO ARRAY [0..0] OF POINTER TO TypeDesc;
	_NUMBEROFMETHODCALLTYPEDESCS : WORD;
	_BSYMBOLSETSACTIVATED : BOOL := FALSE;
	_HRUNTIMEINTERFACE : SysTypes.RTS_IEC_HANDLE := SysTypes.RTS_INVALID_HANDLE;
	_OBJECT : STRING;
	_OBJECTSET : BOOL;
	_HUSERCHANGEEVENT : RTS_IEC_HANDLE;
	_HCALLBACK : RTS_IEC_HANDLE;
	NODEFINDER : SymbolicVarNodeFinder;
	_BFROMUAINFORMATIONMODEL : BOOL := FALSE;
	CHECKINSTANCEACCESSRIGHTS : BOOL;
	FROMUAINFORMATIONMODEL : BOOL;
	RUNTIMEINTERFACE : RTS_IEC_HANDLE;
	SYMBOLCONFIGCRC : UDINT;
	SYMBOLCONFIGNUMOFTYPES : DINT;
	SYMBOLCONFIGTYPELIST : POINTER TO ARRAY [0..0] OF POINTER TO TypeDesc;
	USERMGROBJECT : STRING;
END_VAR
END_FUNCTION_BLOCK

METHOD GETSYMBOLSSETMASK : DWORD
VAR_INPUT
	VARINFO : POINTER TO VariableInformationStruct;
	HUSER : RTS_IEC_HANDLE := RTS_INVALID_HANDLE;
END_VAR
END_METHOD

METHOD GETUSERACCESSRIGHTS : BYTE
VAR_INPUT
	VARINFO : POINTER TO VariableInformationStruct;
	HUSER : RTS_IEC_HANDLE := RTS_INVALID_HANDLE;
END_VAR
END_METHOD

METHOD INITIALIZE : BOOL
VAR_INPUT
	PROOTNODES : POINTER TO ARRAY [0..0] OF POINTER TO SymbolsBaseNode;
	INODECOUNT : DINT;
	PTYPELIST : POINTER TO ARRAY [0..0] OF POINTER TO TypeDesc;
	INUMOFTYPES : DINT;
	CALLEXECUTORFUNCTION : POINTER TO POINTER TO BYTE;
	METHODCALLTYPEDESCS : POINTER TO ARRAY [0..0] OF POINTER TO TypeDesc;
	NUMBEROFMETHODCALLTYPEDESCS : WORD;
	HRUNTIMEINTERFACE : RTS_IEC_HANDLE;
	BSYMBOLSETSACTIVATED : BOOL;
END_VAR
END_METHOD

METHOD INVALIDATESYMBOLS : SysTypes.RTS_IEC_RESULT
END_METHOD

METHOD NODEISHIDDEN : BOOL
VAR_INPUT
	PNODE : IBaseTreeNode;
END_VAR
END_METHOD

METHOD VALIDATESYMBOLS : SysTypes.RTS_IEC_RESULT
END_METHOD

METHOD BROWSEDOWN : IecVarAccess_Interfaces.IBaseTreeNode
VAR_INPUT
	PNODE : IecVarAccess_Interfaces.ICollections.IBaseTreeNode;
	PVARIABLEINFORMATION : POINTER TO IecVarAccess_Interfaces.VariableInformationStruct2;
	BBROWSEINTOCOMPLEXTYPES : BOOL;
	PRESULT : POINTER TO IecVarAccess_Interfaces.SysTypes.RTS_IEC_RESULT;
END_VAR
END_METHOD

METHOD BROWSEGETCHILDBYINDEX : IecVarAccess_Interfaces.IBaseTreeNode
VAR_INPUT
	PNODE : IecVarAccess_Interfaces.IBaseTreeNode;
	DIINDEX : DINT;
	PVARIABLEINFORMATION : POINTER TO IecVarAccess_Interfaces.VariableInformationStruct2;
	PRESULT : POINTER TO UDINT;
END_VAR
END_METHOD

METHOD BROWSEGETNEXT : IecVarAccess_Interfaces.ICollections.IBaseTreeNode
VAR_INPUT
	PNODE : IecVarAccess_Interfaces.ICollections.IBaseTreeNode;
	PVARIABLEINFORMATION : POINTER TO IecVarAccess_Interfaces.VariableInformationStruct2;
	BBROWSEINTOCOMPLEXTYPES : BOOL;
	PRESULT : POINTER TO IecVarAccess_Interfaces.SysTypes.RTS_IEC_RESULT;
END_VAR
END_METHOD

METHOD BROWSEGETROOT : IecVarAccess_Interfaces.IBaseTreeNode
VAR_INPUT
	HUSER : IecVarAccess_Interfaces.RTS_IEC_HANDLE;
	PRESULT : POINTER TO UDINT;
END_VAR
END_METHOD

METHOD BROWSERECURSIVE : SysTypes.RTS_IEC_RESULT
VAR_INPUT
	PNODE : ICollections.IBaseTreeNode;
	PVARIABLEINFORMATION : POINTER TO IecVarAccess_Interfaces.VariableInformationStruct3;
	PFBROWSECALLBACK : POINTER TO BYTE;
	PUSERPARAMETER : POINTER TO BYTE;
END_VAR
END_METHOD

METHOD BROWSEUP : ICollections.IBaseTreeNode
VAR_INPUT
	PNODE : ICollections.IBaseTreeNode;
	PVARIABLEINFORMATION : POINTER TO IecVarAccess_Interfaces.VariableInformationStruct2;
	BBROWSEINTOCOMPLEXTYPES : BOOL;
	PRESULT : POINTER TO IecVarAccess_Interfaces.SysTypes.RTS_IEC_RESULT;
END_VAR
END_METHOD

METHOD DOBROWSEDOWN : ITreeWalker
VAR_INPUT
	PNODE : IecVarAccess_Interfaces.ICollections.IBaseTreeNode;
	PVARIABLEINFORMATION : POINTER TO IecVarAccess_Interfaces.VariableInformationStruct2;
	BBROWSEINTOCOMPLEXTYPES : BOOL;
	PRESULT : POINTER TO IecVarAccess_Interfaces.SysTypes.RTS_IEC_RESULT;
	SYMBOLSET : DWORD;
	USERACCESSRIGHTS : BYTE;
END_VAR
END_METHOD

METHOD DOBROWSENEXT : ITreeWalker
VAR_INPUT
	PNODE : IecVarAccess_Interfaces.ICollections.IBaseTreeNode;
	PVARIABLEINFORMATION : POINTER TO IecVarAccess_Interfaces.VariableInformationStruct2;
	BBROWSEINTOCOMPLEXTYPES : BOOL;
	PRESULT : POINTER TO IecVarAccess_Interfaces.SysTypes.RTS_IEC_RESULT;
	SYMBOLSET : DWORD;
	USERACCESSRIGHTS : BYTE;
END_VAR
END_METHOD

METHOD DOBROWSEUP : ITreeWalker
VAR_INPUT
	PNODE : ICollections.IBaseTreeNode;
	PVARIABLEINFORMATION : POINTER TO IecVarAccess_Interfaces.VariableInformationStruct2;
	BBROWSEINTOCOMPLEXTYPES : BOOL;
	PRESULT : POINTER TO IecVarAccess_Interfaces.SysTypes.RTS_IEC_RESULT;
	SYMBOLSET : DWORD;
	USERACCESSRIGHTS : BYTE;
END_VAR
END_METHOD

METHOD FINDCHILDBYNAME : IecVarAccess_Interfaces.IBaseTreeNode
VAR_INPUT
	PNODE : IecVarAccess_Interfaces.IBaseTreeNode;
	PVARIABLEINFORMATION : POINTER TO IecVarAccess_Interfaces.VariableInformationStruct3;
	PNAME : POINTER TO STRING;
	PRESULT : POINTER TO UDINT;
END_VAR
END_METHOD

METHOD GETNODE : ICollections.IBaseTreeNode
VAR_INPUT
	PSZPATH : POINTER TO STRING;
	PVARIABLEINFORMATION : POINTER TO VariableInformationStruct;
	XRESOLVEBROWSEINFO : BOOL;
	PRESULT : POINTER TO RTS_IEC_RESULT;
END_VAR
END_METHOD

METHOD FB_EXIT : BOOL
VAR_INPUT
	BINCOPYCODE : BOOL;
END_VAR
END_METHOD

METHOD FB_INIT : BOOL
VAR_INPUT
	BINITRETAINS : BOOL;
	BINCOPYCODE : BOOL;
END_VAR
END_METHOD

METHOD FB_REINIT : BOOL
END_METHOD

METHOD EVENTCALLBACK : RTS_IEC_RESULT
VAR_INPUT
	PEVENTPARAM : POINTER TO CmpEventMgr.EventParam;
END_VAR
END_METHOD

METHOD VARACCGETNODEFULLPATH4 : DINT
VAR_INPUT
	PNODE : ICollections.IBaseTreeNode;
	PVARIABLEINFORMATION : POINTER TO IecVarAccess_Interfaces.VariableInformationStruct3;
	PSZPATH : POINTER TO STRING;
	DIMAXPATH : DINT;
	PRESULT : POINTER TO SysTypes.RTS_IEC_RESULT;
END_VAR
END_METHOD

METHOD VARACCGETNODENAME4 : SysTypes.RTS_IEC_RESULT
VAR_INPUT
	PNODE : ICollections.IBaseTreeNode;
	PVARIABLEINFORMATION : POINTER TO IecVarAccess_Interfaces.VariableInformationStruct3;
	PSZNODENAME : POINTER TO STRING;
	NNODENAMELEN : UDINT;
END_VAR
END_METHOD

METHOD BROWSEDOWNINTERNAL : ITreeWalker
VAR_INPUT
	PNODE : ITreeWalker;
	USERACCESSRIGHTS : BYTE;
	SYMBOLSET : DWORD;
	PRESULT : POINTER TO UDINT;
END_VAR
END_METHOD

METHOD BROWSEGETNEXTINTERNAL : ITreeWalker
VAR_INPUT
	PNODE : ITreeWalker;
	USERACCESSRIGHTS : BYTE;
	SYMBOLSET : DWORD;
	PRESULT : POINTER TO UDINT;
END_VAR
END_METHOD

METHOD BROWSEUPINTERNAL : ITreeWalker
VAR_INPUT
	PNODE : ITreeWalker;
	USERACCESSRIGHTS : BYTE;
	SYMBOLSET : DWORD;
	PRESULT : POINTER TO UDINT;
END_VAR
END_METHOD

METHOD ISMEMBER : BOOL
VAR_INPUT
	ITYPENODE : ITypeDesc;
	PNODE : ITreeWalker;
END_VAR
END_METHOD

METHOD RESOLVENODE : RTS_IEC_RESULT
VAR_INPUT
	PNODE : ITreeWalker;
	PVARIABLEINFORMATION : POINTER TO VariableInformationStruct3;
	VARINFOIMPL : REFERENCE TO VariableInformation;
	HANDLEBROWSEINFO : BOOL;
END_VAR
END_METHOD

METHOD EXECUTECALL : RTS_IEC_RESULT
VAR_INPUT
	PNODE : IBaseTreeNode;
	PVARIABLEINFORMATION : POINTER TO VariableInformationStruct;
	PARGUMENTBUFFER : POINTER TO BYTE;
	NARGUMENTBUFFERSIZE : __XWORD;
END_VAR
END_METHOD

METHOD GETVALUE : __XWORD
VAR_INPUT
	PNODE : IBaseTreeNode;
	PVARIABLEINFORMATION : POINTER TO VariableInformationStruct;
	PDEST : POINTER TO BYTE;
	DWSIZE : __XWORD;
	PRESULT : POINTER TO RTS_IEC_RESULT;
END_VAR
END_METHOD

METHOD SETVALUE : __XWORD
VAR_INPUT
	PNODE : IBaseTreeNode;
	PVARIABLEINFORMATION : POINTER TO VariableInformationStruct;
	PSRC : POINTER TO BYTE;
	DWSIZE : __XWORD;
	PRESULT : POINTER TO RTS_IEC_RESULT;
END_VAR
END_METHOD

METHOD SWAPVALUE : __XWORD
VAR_INPUT
	PNODE : IBaseTreeNode;
	PVARIABLEINFORMATION : POINTER TO VariableInformationStruct;
	PDATA : POINTER TO BYTE;
	BMOTOROLA : BOOL;
	PRESULT : POINTER TO RTS_IEC_RESULT;
END_VAR
END_METHOD

METHOD GETACCESSRIGHTS : IecVarAccess_Interfaces.AccessRights
VAR_INPUT
	PNODE : IecVarAccess_Interfaces.IBaseTreeNode;
	PVARIABLEINFORMATION : POINTER TO IecVarAccess_Interfaces.VariableInformationStruct2;
	BGETUSERRIGHTS : BOOL;
	PRESULT : POINTER TO UDINT;
END_VAR
END_METHOD

METHOD GETADDRESS : POINTER TO BYTE
VAR_INPUT
	PNODE : IBaseTreeNode;
	PVARIABLEINFORMATION : POINTER TO VariableInformationStruct;
	PRESULT : POINTER TO RTS_IEC_RESULT;
END_VAR
END_METHOD

METHOD GETATTRIBUTEBYINDEX : POINTER TO STRING
VAR_INPUT
	PNODE : IBaseTreeNode;
	WINDEX : WORD;
	PRESULT : POINTER TO SysTypes.RTS_IEC_RESULT;
END_VAR
END_METHOD

METHOD GETCLIENTOFFSET : __XWORD
VAR_INPUT
	PNODE : IBaseTreeNode;
	PRESULT : POINTER TO SysTypes.RTS_IEC_RESULT;
END_VAR
END_METHOD

METHOD GETNAMESPACENODEFLAGS : IecVarAccess_Interfaces.NamespaceNodeFlags
VAR_INPUT
	PNODE : IBaseTreeNode;
	PRESULT : POINTER TO UDINT;
END_VAR
END_METHOD

METHOD GETNODEFLAGS : DWORD
VAR_INPUT
	PNODE : IBaseTreeNode;
	PRESULT : POINTER TO SysTypes.RTS_IEC_RESULT;
END_VAR
END_METHOD

METHOD GETNODEFULLPATH : DINT
VAR_INPUT
	PNODE : IBaseTreeNode;
	PVARIABLEINFORMATION : POINTER TO VariableInformationStruct;
	PSZPATH : POINTER TO STRING;
	DIMAXPATH : DINT;
	PRESULT : POINTER TO RTS_IEC_RESULT;
END_VAR
END_METHOD

METHOD GETNODENAME : POINTER TO STRING
VAR_INPUT
	PNODE : IBaseTreeNode;
	PVARIABLEINFORMATION : POINTER TO VariableInformationStruct;
	PRESULT : POINTER TO RTS_IEC_RESULT;
END_VAR
END_METHOD

METHOD GETNODETYPE : TreeNodeType
VAR_INPUT
	PNODE : IBaseTreeNode;
	PRESULT : POINTER TO UDINT;
END_VAR
END_METHOD

METHOD GETNUMOFATTRIBUTES : WORD
VAR_INPUT
	PNODE : IBaseTreeNode;
	PRESULT : POINTER TO SysTypes.RTS_IEC_RESULT;
END_VAR
END_METHOD

METHOD GETSIZE : __XWORD
VAR_INPUT
	PNODE : IBaseTreeNode;
	PVARIABLEINFORMATION : POINTER TO VariableInformationStruct;
	PRESULT : POINTER TO RTS_IEC_RESULT;
END_VAR
END_METHOD

METHOD GETSWAPSIZE : __XWORD
VAR_INPUT
	PNODE : IBaseTreeNode;
	PRESULT : POINTER TO RTS_IEC_RESULT;
END_VAR
END_METHOD

METHOD GETTYPECLASS : TypeClass
VAR_INPUT
	PNODE : IBaseTreeNode;
	PVARIABLEINFORMATION : POINTER TO VariableInformationStruct;
	PRESULT : POINTER TO RTS_IEC_RESULT;
END_VAR
END_METHOD

METHOD GETTYPENODE : ITypeDesc
VAR_INPUT
	PNODE : IBaseTreeNode;
	PVARIABLEINFORMATION : POINTER TO VariableInformationStruct;
	PRESULT : POINTER TO RTS_IEC_RESULT;
	OPTIONS : WORD := GetTypeNodeOptions.GetBaseType;
END_VAR
END_METHOD

METHOD ISREFERENCE : BOOL
VAR_INPUT
	PNODE : IBaseTreeNode;
	PVARIABLEINFORMATION : POINTER TO VariableInformationStruct;
	PRESULT : POINTER TO RTS_IEC_RESULT;
END_VAR
END_METHOD

METHOD GETCHILDBYBROWSENAME : IBaseTreeNode
VAR_INPUT
	HNODE : RTS_IEC_HANDLE;
	PVARIABLEINFORMATION : POINTER TO IecVarAccess_Interfaces.VariableInformationStruct2;
	PBROWSENAME : POINTER TO OpcUa_QualifiedName;
	PRESULT : POINTER TO UDINT;
END_VAR
END_METHOD

METHOD GETNEXTBYBROWSENAME : IBaseTreeNode
VAR_INPUT
	HNODE : RTS_IEC_HANDLE;
	PVARIABLEINFORMATION : POINTER TO IecVarAccess_Interfaces.VariableInformationStruct2;
	PBROWSENAME : POINTER TO OpcUa_QualifiedName;
	PRESULT : POINTER TO UDINT;
END_VAR
END_METHOD

METHOD GETBROWSENAME : SysTypes.RTS_IEC_RESULT
VAR_INPUT
	HNODE : RTS_IEC_HANDLE;
END_VAR
VAR_OUTPUT
	PBROWSENAME : POINTER TO CmpOPCUAStack_Interfaces.OpcUa_QualifiedName;
END_VAR
END_METHOD

METHOD GETDESCRIPTION : SysTypes.RTS_IEC_RESULT
VAR_INPUT
	HNODE : RTS_IEC_HANDLE;
END_VAR
VAR_OUTPUT
	PDESCRIPTION : POINTER TO CmpOPCUAStack_Interfaces.OpcUa_LocalizedText;
END_VAR
END_METHOD

METHOD GETDISPLAYNAME : SysTypes.RTS_IEC_RESULT
VAR_INPUT
	HNODE : RTS_IEC_HANDLE;
END_VAR
VAR_OUTPUT
	PDISPLAYNAME : POINTER TO CmpOPCUAStack_Interfaces.OpcUa_LocalizedText;
END_VAR
END_METHOD

METHOD GETENTRYPOINT : RTS_IEC_RESULT
VAR_INPUT
	HNODE : RTS_IEC_HANDLE;
END_VAR
VAR_OUTPUT
	ISENTRYPOINT : BOOL;
	PENTRYPOINT : POINTER TO CmpOPCUAStack_Interfaces.OpcUa_NodeId;
END_VAR
END_METHOD

METHOD GETEVENTNOTIFIER : SysTypes.RTS_IEC_RESULT
VAR_INPUT
	HNODE : RTS_IEC_HANDLE;
END_VAR
VAR_OUTPUT
	EVENTNOTIFIER : CmpOPCUAStack_Interfaces.OpcUa_Byte;
END_VAR
END_METHOD

METHOD GETMETHODARGUMENTS : RTS_IEC_RESULT
VAR_INPUT
	HNODE : RTS_IEC_HANDLE;
END_VAR
VAR_OUTPUT
	PINPUTARGUMENTS : POINTER TO OpcUa_NodeId;
	POUTPUTARGUMENTS : POINTER TO OpcUa_NodeId;
END_VAR
END_METHOD

METHOD GETNODECLASS : SysTypes.RTS_IEC_RESULT
VAR_INPUT
	HNODE : RTS_IEC_HANDLE;
END_VAR
VAR_OUTPUT
	NODECLASS : CmpOPCUAStack_Interfaces.OpcUa_NodeClass;
END_VAR
END_METHOD

METHOD GETPARENTREFERENCETYPE : SysTypes.RTS_IEC_RESULT
VAR_INPUT
	HNODE : RTS_IEC_HANDLE;
END_VAR
VAR_OUTPUT
	PREFERENCETYPE : POINTER TO OpcUa_NodeId;
END_VAR
END_METHOD

METHOD GETTYPEDEFINITION : SysTypes.RTS_IEC_RESULT
VAR_INPUT
	HNODE : RTS_IEC_HANDLE;
END_VAR
VAR_OUTPUT
	PTYPEDEFINITION : POINTER TO OpcUa_NodeId;
END_VAR
END_METHOD

METHOD TYPEGETDATATYPEID : RTS_IEC_RESULT
VAR_INPUT
	HTYPENODE : RTS_IEC_HANDLE;
END_VAR
VAR_OUTPUT
	PDATATYPEID : POINTER TO OpcUa_NodeId;
END_VAR
END_METHOD

METHOD TYPEGETENCODINGNODEID : RTS_IEC_RESULT
VAR_INPUT
	HTYPENODE : RTS_IEC_HANDLE;
END_VAR
VAR_OUTPUT
	PENCODINGID : POINTER TO OpcUa_NodeId;
END_VAR
END_METHOD

METHOD TYPEGETPARENTNODE : RTS_IEC_RESULT
VAR_INPUT
	HTYPENODE : RTS_IEC_HANDLE;
END_VAR
VAR_OUTPUT
	PPARENTNODE : POINTER TO OpcUa_NodeId;
END_VAR
END_METHOD

METHOD TYPEGETPARENTREFERENCETYPE : RTS_IEC_RESULT
VAR_INPUT
	HTYPENODE : RTS_IEC_HANDLE;
END_VAR
VAR_OUTPUT
	PPARENTREFERENCETYPE : POINTER TO OpcUa_NodeId;
END_VAR
END_METHOD

METHOD TYPEISWELLKNOWNTYPE : RTS_IEC_RESULT
VAR_INPUT
	HTYPENODE : RTS_IEC_HANDLE;
END_VAR
VAR_OUTPUT
	TYPEWELLKNOWN : BOOL;
END_VAR
END_METHOD

METHOD GETBASETYPE : ITypeDesc
VAR_INPUT
	TYPEDESC : ITypeDesc;
END_VAR
END_METHOD

METHOD GETENUMMEMBERATTRIBUTELIST : POINTER TO EnumAttributes
VAR_INPUT
	TYPEDESC : ITypeDesc;
	PNNUMOFENUMVALUES : POINTER TO INT;
	PRESULT : POINTER TO SysTypes.RTS_IEC_RESULT;
END_VAR
END_METHOD

METHOD GETENUMVALUES : POINTER TO EnumValues
VAR_INPUT
	TYPEDESC : ITypeDesc;
	PNNUMOFENUMVALUES : POINTER TO INT;
	PRESULT : POINTER TO SysTypes.RTS_IEC_RESULT;
END_VAR
END_METHOD

METHOD GETNUMOFTYPEATTRIBUTES : WORD
VAR_INPUT
	TYPEDESC : ITypeDesc;
	PRESULT : POINTER TO SysTypes.RTS_IEC_RESULT;
END_VAR
END_METHOD

METHOD GETNUMOFTYPES : DINT
VAR_INPUT
	PRESULT : POINTER TO SysTypes.RTS_IEC_RESULT;
END_VAR
END_METHOD

METHOD GETRANGE : BOOL
VAR_INPUT
	TYPEDESC : ITypeDesc;
	PLOWER : POINTER TO LWORD;
	PUPPER : POINTER TO LWORD;
	PRESULT : POINTER TO SysTypes.RTS_IEC_RESULT;
END_VAR
END_METHOD

METHOD GETREFERENCEBASETYPE : ITypeDesc
VAR_INPUT
	TYPEDESC : ITypeDesc;
	PRESULT : POINTER TO SysTypes.RTS_IEC_RESULT;
END_VAR
END_METHOD

METHOD GETTYPEATTRIBUTEBYINDEX : POINTER TO STRING
VAR_INPUT
	TYPEDESC : ITypeDesc;
	WINDEX : WORD;
	PRESULT : POINTER TO SysTypes.RTS_IEC_RESULT;
END_VAR
END_METHOD

METHOD GETTYPECLASSFROMTYPE : TypeClass
VAR_INPUT
	TYPEDESC : ITypeDesc;
	DWFLAGS : DWORD;
	PRESULT : POINTER TO RTS_IEC_RESULT;
END_VAR
END_METHOD

METHOD GETTYPEDESC : UDINT
VAR_INPUT
	PTYPEDESC : ITypeDesc;
	PTYPEDESCSTRUCT : POINTER TO TypeDescAsUnion;
END_VAR
END_METHOD

METHOD GETTYPEDESCVARLENARRAY : RTS_IEC_RESULT
VAR_INPUT
	PTYPEDESC : ITypeDesc;
	PTYPEDESCSTRUCT : POINTER TO TypeDescVarArrayAsStruct;
END_VAR
END_METHOD

METHOD GETTYPENAME : POINTER TO STRING
VAR_INPUT
	TYPEDESC : ITypeDesc;
	PRESULT : POINTER TO SysTypes.RTS_IEC_RESULT;
END_VAR
END_METHOD

METHOD GETTYPENODEBYINDEX : ITypeDesc
VAR_INPUT
	DIINDEX : DINT;
	PRESULT : POINTER TO SysTypes.RTS_IEC_RESULT;
END_VAR
END_METHOD

METHOD GETUABUILTINTYPE : USINT
VAR_INPUT
	TYPEDESC : ITypeDesc;
	PRESULT : POINTER TO RTS_IEC_RESULT;
END_VAR
END_METHOD

METHOD HASBASETYPE : BOOL
VAR_INPUT
	TYPEDESC : ITypeDesc;
END_VAR
END_METHOD

METHOD EXITVARINFO : SysTypes.RTS_IEC_RESULT
VAR_INPUT
	PVARIABLEINFORMATION : POINTER TO IecVarAccess_Interfaces.VariableInformationStruct2;
END_VAR
END_METHOD

METHOD INITVARINFO : IecVarAccess_Interfaces.SysTypes.RTS_IEC_RESULT
VAR_INPUT
	PVARIABLEINFORMATION : POINTER TO IecVarAccess_Interfaces.VariableInformationStruct2;
	NSIZEOFVARINFO : UINT;
	HUSER : IecVarAccess_Interfaces.RTS_IEC_HANDLE;
END_VAR
END_METHOD

(* ---- SYMBOLICVARNODEFINDER.pou ---- *)
FUNCTION_BLOCK SYMBOLICVARNODEFINDER
VAR
	_ROOTNODES : POINTER TO ARRAY [0..0] OF POINTER TO SymbolsBaseNode;
	_ROOTNODECOUNT : DINT;
	_SEARCHCALLBACKS : ISearchCallbacks;
	NAME : POINTER TO STRING;
END_VAR
END_FUNCTION_BLOCK

METHOD FINDLONGWITHDATA : ITreeWalker
VAR_INPUT
	PSTPATH : POINTER TO STRING;
	VARINFO : REFERENCE TO VariableInformation;
	VIEW : DWORD;
END_VAR
VAR_OUTPUT
	BEND : BOOL;
	PRT : POINTER TO IInstancePathBuildingNode;
END_VAR
END_METHOD

METHOD GETSYMBOLICNODE : ITreeWalker
VAR_INPUT
	PSZPATH : POINTER TO BYTE;
	VARIABLEINFO : REFERENCE TO VariableInformation;
	VIEW : DWORD;
	PRESULT : POINTER TO UDINT;
END_VAR
END_METHOD

METHOD GETSYMBOLICSUBNODE : ITreeWalker
VAR_INPUT
	PSZPATH : POINTER TO BYTE;
	OFFSETINPATH : __XWORD;
	CURRENTNODE : ITreeWalker;
	VIEW : DWORD;
	PRESULT : POINTER TO UDINT;
END_VAR
VAR_IN_OUT
	VARIABLEINFO : VariableInformation;
END_VAR
END_METHOD

METHOD INITIALIZE : BOOL
VAR_INPUT
	PROOTNODES : POINTER TO ARRAY [0..0] OF POINTER TO SymbolsBaseNode;
	INODECOUNT : DINT;
END_VAR
END_METHOD

METHOD INITIALIZE2 : BOOL
VAR_INPUT
	PROOTNODES : POINTER TO ARRAY [0..0] OF POINTER TO SymbolsBaseNode;
	INODECOUNT : DINT;
	CALLBACKS : ISearchCallbacks;
END_VAR
END_METHOD

METHOD ASBASETREENODE : ICollections.IBaseTreeNode
END_METHOD

METHOD FINDCHILD : ITreeWalker
VAR_INPUT
	SZCHILDNAME : POINTER TO BYTE;
	NAMELEN : __XWORD;
	SYMBOLSSETS : DWORD;
	VARINFO : REFERENCE TO VariableInformation;
	PRESULT : POINTER TO RTS_IEC_RESULT;
END_VAR
VAR_IN_OUT
	TYPESYSTEMREACHED : BOOL;
END_VAR
END_METHOD

METHOD GETCHILDBYINDEX : ITreeWalker
VAR_INPUT
	IINDEX : DINT;
	USERACCESSRIGHTS : BYTE;
	SYMBOLSSETS : DWORD;
END_VAR
VAR_OUTPUT
	XOUTOFRANGE : BOOL;
END_VAR
END_METHOD

METHOD GETFIRSTCHILD : ITreeWalker
VAR_INPUT
	USERACCESSRIGHTS : BYTE;
	SYMBOLSSETS : DWORD;
END_VAR
END_METHOD

METHOD GETFULLPATH : DINT
VAR_INPUT
	PBUFFER : POINTER TO STRING;
	DIBUFFERSIZE : DINT;
END_VAR
VAR_OUTPUT
	BROOT_NODE : BOOL;
	BEMPTYNAMESPACENODE : BOOL;
END_VAR
END_METHOD

METHOD GETPARENT : ITreeWalker
VAR_INPUT
	USERACCESSRIGHTS : BYTE;
	SYMBOLSSETS : DWORD;
END_VAR
END_METHOD

METHOD GETSIBLING : ITreeWalker
VAR_INPUT
	USERACCESSRIGHTS : BYTE;
	SYMBOLSSETS : DWORD;
END_VAR
END_METHOD

METHOD ISVISIBLE : BOOL
VAR_INPUT
	USERACCESSRIGHTS : BYTE;
	SYMBOLSSETS : DWORD;
END_VAR
END_METHOD

METHOD FINDNODE : ITreeWalker
VAR_INPUT
	PSTPATH : POINTER TO STRING;
	VIEW : DWORD;
	STARTPOS : __XWORD;
	OPTEXPLICITCURRENTNODE : ITreeWalker;
END_VAR
VAR_OUTPUT
	BEND : BOOL;
	PRT : POINTER TO IInstancePathBuildingNode;
END_VAR
VAR_IN_OUT
	VARINFO : VariableInformation;
END_VAR
END_METHOD

METHOD HANDLEGETSYMBOLICNODERESULT : ITreeWalker
VAR_INPUT
	PFIND : ITreeWalker;
	PRESULT : POINTER TO UDINT;
END_VAR
END_METHOD

METHOD GETCHILDBYBROWSENAME : ITreeWalker
VAR_INPUT
	PBROWSENAME : POINTER TO OpcUa_QualifiedName;
	VARINFO : REFERENCE TO VariableInformation;
END_VAR
END_METHOD

METHOD GETNEXTBYBROWSENAME : ITreeWalker
VAR_INPUT
	PBROWSENAME : POINTER TO OpcUa_QualifiedName;
	VARINFO : REFERENCE TO VariableInformation;
END_VAR
END_METHOD

(* ---- SYMBOLSBASENODE.pou ---- *)
FUNCTION_BLOCK SYMBOLSBASENODE
VAR
	_FATHER : POINTER TO SymbolsBaseNode;
	_ICOUNT : DINT;
	_PSTNAME : POINTER TO STRING;
	_DWSYMBOLSETMASK : DWORD := ANY_TO_DWORD(-1);
	_INDEX : DINT := -1;
	_TYPE : InstancePathBuildingNodeType;
	_IBASETREENODE : IBaseTreeNode := THIS^;
	_IMEMBERINDEX : IMemberIndex := THIS^;
	_ITREEWALKER : ITreeWalker := THIS^;
	_OPCUAMETADATA : REFERENCE TO OpcUaNodeMetaData;
	CHILDCOUNT : DINT;
	ISSTATICVARWITHINNONSTATICFBINSTANCE : BOOL;
	MEMBERINDEX : DINT;
	NAME : POINTER TO STRING;
	NUMCHILDS : DINT;
	PROCHILDREN : POINTER TO ARRAY [0..100] OF ICollections.IBaseTreeNode;
END_VAR
END_FUNCTION_BLOCK

METHOD ADDREF : DINT
END_METHOD

METHOD FB_EXIT : BOOL
VAR_INPUT
	BINCOPYCODE : BOOL;
END_VAR
END_METHOD

METHOD FB_INIT : BOOL
VAR_INPUT
	BINITRETAINS : BOOL;
	BINCOPYCODE : BOOL;
END_VAR
END_METHOD

METHOD FB_REINIT : BOOL
END_METHOD

METHOD QUERYINTERFACE : POINTER TO POINTER TO BYTE
VAR_INPUT
	IID : DWORD;
	PRESULT : POINTER TO UDINT;
END_VAR
END_METHOD

METHOD RELEASE : DINT
END_METHOD

METHOD GETCHILD : ICollections.IBaseTreeNode
VAR_INPUT
	DIINDEX : DINT;
END_VAR
END_METHOD

METHOD GETFATHER : ICollections.IBaseTreeNode
END_METHOD

METHOD GETBROWSENAME : SysTypes.RTS_IEC_RESULT
VAR_OUTPUT
	PBROWSENAME : POINTER TO CmpOPCUAStack_Interfaces.OpcUa_QualifiedName;
END_VAR
END_METHOD

METHOD GETDESCRIPTION : SysTypes.RTS_IEC_RESULT
VAR_OUTPUT
	PDESCRIPTION : POINTER TO CmpOPCUAStack_Interfaces.OpcUa_LocalizedText;
END_VAR
END_METHOD

METHOD GETDISPLAYNAME : SysTypes.RTS_IEC_RESULT
VAR_OUTPUT
	PDISPLAYNAME : POINTER TO CmpOPCUAStack_Interfaces.OpcUa_LocalizedText;
END_VAR
END_METHOD

METHOD GETENTRYPOINT : RTS_IEC_RESULT
VAR_OUTPUT
	ISENTRYPOINT : BOOL;
	PENTRYPOINT : POINTER TO CmpOPCUAStack_Interfaces.OpcUa_NodeId;
END_VAR
END_METHOD

METHOD GETEVENTNOTIFIER : SysTypes.RTS_IEC_RESULT
VAR_OUTPUT
	EVENTNOTIFIER : CmpOPCUAStack_Interfaces.OpcUa_Byte;
END_VAR
END_METHOD

METHOD GETNODECLASS : SysTypes.RTS_IEC_RESULT
VAR_OUTPUT
	NODECLASS : CmpOPCUAStack_Interfaces.OpcUa_NodeClass;
END_VAR
END_METHOD

METHOD GETPARENTREFERENCETYPE : SysTypes.RTS_IEC_RESULT
VAR_OUTPUT
	PREFERENCETYPE : POINTER TO OpcUa_NodeId;
END_VAR
END_METHOD

METHOD GETTYPEDEFINITION : SysTypes.RTS_IEC_RESULT
VAR_OUTPUT
	PTYPEDEFINITION : POINTER TO OpcUa_NodeId;
END_VAR
END_METHOD

METHOD ASBASETREENODE : ICollections.IBaseTreeNode
END_METHOD

METHOD FINDCHILD : ITreeWalker
VAR_INPUT
	SZCHILDNAME : POINTER TO BYTE;
	NAMELEN : __XWORD;
	SYMBOLSSETS : DWORD;
	VARINFO : REFERENCE TO VariableInformation;
	PRESULT : POINTER TO RTS_IEC_RESULT;
END_VAR
VAR_IN_OUT
	TYPESYSTEMREACHED : BOOL;
END_VAR
END_METHOD

METHOD GETCHILDBYINDEX : ITreeWalker
VAR_INPUT
	IINDEX : DINT;
	USERACCESSRIGHTS : BYTE;
	SYMBOLSSETS : DWORD;
END_VAR
VAR_OUTPUT
	XOUTOFRANGE : BOOL;
END_VAR
END_METHOD

METHOD GETFIRSTCHILD : ITreeWalker
VAR_INPUT
	USERACCESSRIGHTS : BYTE;
	SYMBOLSSETS : DWORD;
END_VAR
END_METHOD

METHOD GETFULLPATH : DINT
VAR_INPUT
	PBUFFER : POINTER TO STRING;
	DIBUFFERSIZE : DINT;
END_VAR
VAR_OUTPUT
	BROOT_NODE : BOOL;
	BEMPTYNAMESPACENODE : BOOL;
END_VAR
END_METHOD

METHOD GETPARENT : ITreeWalker
VAR_INPUT
	USERACCESSRIGHTS : BYTE;
	SYMBOLSSETS : DWORD;
END_VAR
END_METHOD

METHOD GETSIBLING : ITreeWalker
VAR_INPUT
	USERACCESSRIGHTS : BYTE;
	SYMBOLSSETS : DWORD;
END_VAR
END_METHOD

METHOD ISVISIBLE : BOOL
VAR_INPUT
	USERACCESSRIGHTS : BYTE;
	SYMBOLSSETS : DWORD;
END_VAR
END_METHOD

METHOD GETBYBROWSENAMEINDEX : ITreeWalker
VAR_INPUT
	PBROWSENAME : POINTER TO OpcUa_QualifiedName;
	VARINFO : REFERENCE TO VariableInformation;
END_VAR
VAR_OUTPUT
	RESULT : RTS_IEC_RESULT;
END_VAR
END_METHOD

METHOD GETCHILDBYBROWSENAME : ITreeWalker
VAR_INPUT
	PBROWSENAME : POINTER TO OpcUa_QualifiedName;
	VARINFO : REFERENCE TO VariableInformation;
END_VAR
END_METHOD

METHOD GETNEXTBYBROWSENAME : ITreeWalker
VAR_INPUT
	PBROWSENAME : POINTER TO OpcUa_QualifiedName;
	VARINFO : REFERENCE TO VariableInformation;
END_VAR
END_METHOD

(* ---- SYMBOLSBRANCHNODE.pou ---- *)
FUNCTION_BLOCK SYMBOLSBRANCHNODE EXTENDS SymbolsBaseNode
VAR
	_PCHILDREN : POINTER TO ARRAY [0..0] OF POINTER TO SymbolsBaseNode;
	_PCHILDRENBYBROWSENAME : POINTER TO POINTER TO SymbolsBaseNode;
	_ICHILDCOUNT : DINT;
	INSTANCEPATHNODETYPE : InstancePathBuildingNodeType;
	MEMBERINDEX : DINT;
	NUMCHILDS : DINT;
END_VAR
END_FUNCTION_BLOCK

METHOD FINDCHILD : ITreeWalker
VAR_INPUT
	SZCHILDNAME : POINTER TO BYTE;
	NAMELEN : __XWORD;
	SYMBOLSSETS : DWORD;
	VARINFO : REFERENCE TO VariableInformation;
	PRESULT : POINTER TO RTS_IEC_RESULT;
END_VAR
VAR_IN_OUT
	TYPESYSTEMREACHED : BOOL;
END_VAR
END_METHOD

METHOD GETBYBROWSENAMEINDEX : ITreeWalker
VAR_INPUT
	PBROWSENAME : POINTER TO OpcUa_QualifiedName;
	VARINFO : REFERENCE TO VariableInformation;
END_VAR
VAR_OUTPUT
	RESULT : RTS_IEC_RESULT;
END_VAR
END_METHOD

METHOD GETCHILDBYBROWSENAME : ITreeWalker
VAR_INPUT
	PBROWSENAME : POINTER TO OpcUa_QualifiedName;
	VARINFO : REFERENCE TO VariableInformation;
END_VAR
END_METHOD

METHOD GETCHILDBYINDEX : ITreeWalker
VAR_INPUT
	IINDEX : DINT;
	USERACCESSRIGHTS : BYTE;
	SYMBOLSSETS : DWORD;
END_VAR
VAR_OUTPUT
	XOUTOFRANGE : BOOL;
END_VAR
END_METHOD

METHOD GETFIRSTCHILD : ITreeWalker
VAR_INPUT
	USERACCESSRIGHTS : BYTE;
	SYMBOLSSETS : DWORD;
END_VAR
END_METHOD

(* ---- TYPEDESC.pou ---- *)
FUNCTION_BLOCK TYPEDESC
VAR
	_DWSIZE : __XWORD;
	_TYPEFLAGS : DWORD;
	_OPCUAMETADATA : REFERENCE TO OpcUaTypeMetaData;
	METHODCALLTYPEINDEX_INTERNAL : WORD;
END_VAR
END_FUNCTION_BLOCK

METHOD BROWSEINTOTYPE : ITreeWalker
VAR_INPUT
	PNODE : ITreeWalker;
	PVARINFO : REFERENCE TO VariableInformation;
	PBROWSEINFO : POINTER TO RtsBrowseInfo;
END_VAR
END_METHOD

METHOD BROWSENEXTELEMENT : ITreeWalker
VAR_INPUT
	PNODE : ITreeWalker;
	PVARINFO : REFERENCE TO VariableInformation;
	PBROWSEINFO : POINTER TO RtsBrowseInfo;
END_VAR
END_METHOD

METHOD BROWSEOUTOFTYPE : ITreeWalker
VAR_INPUT
	PNODE : ITreeWalker;
	PVARINFO : REFERENCE TO VariableInformation;
	PBROWSEINFO : POINTER TO RtsBrowseInfo;
END_VAR
END_METHOD

METHOD EXECUTE_INTERNAL : RTS_IEC_RESULT
VAR_INPUT
	VARINFO : REFERENCE TO VariableInformation;
	PINST : POINTER TO BYTE;
	PMETHODPARAMS : POINTER TO BYTE;
	METHODPRAMSSIZE : __XWORD;
END_VAR
END_METHOD

METHOD FINDCHILD : ITreeWalker
VAR_INPUT
	PSTPATH : POINTER TO STRING;
	VARINFO : REFERENCE TO VariableInformation;
	PRESULT : POINTER TO UDINT;
END_VAR
VAR_IN_OUT
	IOFFSETINPATH : __XWORD;
END_VAR
END_METHOD

METHOD FINDNODE_INTERNAL : IecVarAccess_Interfaces.IInstancePathBuildingNode
VAR_INPUT
	PSTPATH : POINTER TO STRING;
	VARINFO : REFERENCE TO VariableInformation;
	PRESULT : POINTER TO UDINT;
END_VAR
VAR_IN_OUT
	IOFFSETINPATH : DINT;
END_VAR
END_METHOD

METHOD GETADDRESS : POINTER TO BYTE
VAR_INPUT
	PADDRESS : POINTER TO BYTE;
	PRESULT : POINTER TO UDINT;
END_VAR
END_METHOD

METHOD GETATTRIBUTEBYINDEX_INTERNAL : POINTER TO STRING
VAR_INPUT
	WINDEX : WORD;
END_VAR
END_METHOD

METHOD GETBASETYPE_INTERNAL : REFERENCE TO TypeDesc
END_METHOD

METHOD GETENUMMEMBERATTRIBUTELIST_INTERNAL : POINTER TO EnumAttributes
VAR_INPUT
	PNNUMOFENUMVALUES : POINTER TO INT;
	PRESULT : POINTER TO RTS_IEC_RESULT;
END_VAR
END_METHOD

METHOD GETENUMVALUES_INTERNAL : POINTER TO EnumValues
VAR_INPUT
	PNNUMOFENUMVALUES : POINTER TO INT;
	PRESULT : POINTER TO RTS_IEC_RESULT;
END_VAR
END_METHOD

METHOD GETNAME_INTERNAL : POINTER TO STRING
VAR_INPUT
	PRESULT : POINTER TO SysTypes.RTS_IEC_RESULT;
END_VAR
END_METHOD

METHOD GETNATIVESIZE2_INTERNAL : __XWORD
VAR_INPUT
	VARINFO : REFERENCE TO VariableInformation;
END_VAR
END_METHOD

METHOD GETNATIVESIZE_INTERNAL : __XWORD
END_METHOD

METHOD GETNUMOFATTRIBUTES_INTERNAL : WORD
END_METHOD

METHOD GETRANGE_INTERNAL : BOOL
VAR_INPUT
	PLOWER : POINTER TO LWORD;
	PUPPER : POINTER TO LWORD;
END_VAR
END_METHOD

METHOD GETREFERENCEBASETYPE_INTERNAL : REFERENCE TO TypeDesc
VAR_INPUT
	PRESULT : POINTER TO RTS_IEC_RESULT;
END_VAR
END_METHOD

METHOD GETSIZE2_INTERNAL : __XWORD
VAR_INPUT
	VARINFO : REFERENCE TO VariableInformation;
END_VAR
END_METHOD

METHOD GETSIZE_INTERNAL : __XWORD
END_METHOD

METHOD GETSWAPSIZE_INTERNAL : __XWORD
END_METHOD

METHOD GETTYPECLASS2_INTERNAL : TypeClass
VAR_INPUT
	DWFLAGS : DWORD;
END_VAR
END_METHOD

METHOD GETTYPECLASS_INTERNAL : TypeClass
END_METHOD

METHOD GETTYPEDESCVARLENARRAY_INTERNAL : RTS_IEC_RESULT
VAR_INPUT
	PTYPEDESCSTRUCT : POINTER TO TypeDescVarArrayAsStruct;
END_VAR
END_METHOD

METHOD GETTYPEDESC_INTERNAL : UDINT
VAR_INPUT
	PTYPEDESCSTRUCT : POINTER TO TypeDescAsUnion;
END_VAR
END_METHOD

METHOD GETTYPENODE_INTERNAL : REFERENCE TO TypeDesc
VAR_INPUT
	VARINFO : REFERENCE TO VariableInformation;
	OPTIONS : WORD;
END_VAR
END_METHOD

METHOD GETUABUILTINTYPE_INTERNAL : OpcUa_BuiltInType
END_METHOD

METHOD GET_INTERNAL : __XWORD
VAR_INPUT
	PDEST : POINTER TO BYTE;
	PSRC : POINTER TO BYTE;
	VARINFO : REFERENCE TO VariableInformation;
	DWSIZE : __XWORD;
	PRESULT : POINTER TO UDINT;
END_VAR
END_METHOD

METHOD ISMEMBER : BOOL
VAR_INPUT
	PNODE : ITreeWalker;
END_VAR
END_METHOD

METHOD NODEFOUND_INTERNAL : UDINT
VAR_INPUT
	VARINFO : REFERENCE TO VariableInformation;
	BDIRECTCHILDFOUND : BOOL;
END_VAR
END_METHOD

METHOD SET_INTERNAL : __XWORD
VAR_INPUT
	PSRC : POINTER TO BYTE;
	PDEST : POINTER TO BYTE;
	VARINFO : REFERENCE TO VariableInformation;
	DWSIZE : __XWORD;
	PRESULT : POINTER TO UDINT;
END_VAR
END_METHOD

METHOD SWAP_INTERNAL : __XWORD
VAR_INPUT
	PDATA : POINTER TO BYTE;
	VARINFO : REFERENCE TO VariableInformation;
	DWSIZE : __XWORD;
	BMOTOROLA : BOOL;
	PRESULT : POINTER TO UDINT;
END_VAR
END_METHOD

METHOD GETFIRSTCHILDBYBROWSENAME : ITreeWalker
VAR_INPUT
	PBROWSENAME : POINTER TO OpcUa_QualifiedName;
	VARINFO : REFERENCE TO VariableInformation;
END_VAR
VAR_OUTPUT
	RESULT : RTS_IEC_RESULT;
END_VAR
END_METHOD

METHOD GETNEXTCHILDBYBROWSENAME : ITreeWalker
VAR_INPUT
	PBROWSENAME : POINTER TO OpcUa_QualifiedName;
	VARINFO : REFERENCE TO VariableInformation;
	PBROWSEINFO : POINTER TO RtsBrowseInfo;
END_VAR
VAR_OUTPUT
	RESULT : RTS_IEC_RESULT;
END_VAR
END_METHOD

METHOD GETDATATYPEID : RTS_IEC_RESULT
VAR_OUTPUT
	PDATATYPEID : POINTER TO OpcUa_NodeId;
END_VAR
END_METHOD

METHOD GETENCODINGNODEID : RTS_IEC_RESULT
VAR_OUTPUT
	PENCODINGID : POINTER TO OpcUa_NodeId;
END_VAR
END_METHOD

METHOD GETMETHODARGUMENTS : SysTypes.RTS_IEC_RESULT
VAR_OUTPUT
	PINPUTARGUMENTS : POINTER TO CmpOPCUAStack_Interfaces.OpcUa_NodeId;
	POUTPUTARGUMENTS : POINTER TO CmpOPCUAStack_Interfaces.OpcUa_NodeId;
END_VAR
END_METHOD

METHOD GETPARENTNODE : RTS_IEC_RESULT
VAR_OUTPUT
	PPARENTNODE : POINTER TO OpcUa_NodeId;
END_VAR
END_METHOD

METHOD GETPARENTREFERENCETYPE : RTS_IEC_RESULT
VAR_OUTPUT
	PPARENTREFERENCETYPE : POINTER TO OpcUa_NodeId;
END_VAR
END_METHOD

METHOD ISWELLKNOWNTYPE : BOOL
END_METHOD

METHOD FINDNODE : IecVarAccess_Interfaces.IInstancePathBuildingNode
VAR_INPUT
	PSTPATH : POINTER TO STRING;
	VARINFO : IecVarAccess_Interfaces.IVariableInformation;
	PRESULT : POINTER TO UDINT;
END_VAR
VAR_IN_OUT
	IOFFSETINPATH : DINT;
END_VAR
END_METHOD

METHOD GET : IecVarAccess_Interfaces.XWORD
VAR_INPUT
	PDEST : POINTER TO BYTE;
	PSRC : POINTER TO BYTE;
	VARINFO : IecVarAccess_Interfaces.IVariableInformation;
	DWSIZE : IecVarAccess_Interfaces.XWORD;
	PRESULT : POINTER TO UDINT;
END_VAR
END_METHOD

METHOD GETNATIVESIZE : IecVarAccess_Interfaces.XWORD
END_METHOD

METHOD GETSIZE : IecVarAccess_Interfaces.XWORD
END_METHOD

METHOD GETSIZE2 : IecVarAccess_Interfaces.XWORD
VAR_INPUT
	VARINFO : IecVarAccess_Interfaces.IVariableInformation;
END_VAR
END_METHOD

METHOD GETSWAPSIZE : IecVarAccess_Interfaces.XWORD
END_METHOD

METHOD GETTYPECLASS : IecVarAccess_Interfaces.TypeClass
END_METHOD

METHOD GETTYPEDESC : UDINT
VAR_INPUT
	PTYPEDESCSTRUCT : POINTER TO IecVarAccess_Interfaces.TypeDescAsUnion;
END_VAR
END_METHOD

METHOD GETTYPENODE : IecVarAccess_Interfaces.ITypeDesc
VAR_INPUT
	VARINFO : IecVarAccess_Interfaces.IVariableInformation;
END_VAR
END_METHOD

METHOD NODEFOUND : UDINT
VAR_INPUT
	VARINFO : IecVarAccess_Interfaces.IVariableInformation;
	BDIRECTCHILDFOUND : BOOL;
END_VAR
END_METHOD

METHOD SET : IecVarAccess_Interfaces.XWORD
VAR_INPUT
	PSRC : POINTER TO BYTE;
	PDEST : POINTER TO BYTE;
	VARINFO : IecVarAccess_Interfaces.IVariableInformation;
	DWSIZE : IecVarAccess_Interfaces.XWORD;
	PRESULT : POINTER TO UDINT;
END_VAR
END_METHOD

METHOD SWAP : IecVarAccess_Interfaces.XWORD
VAR_INPUT
	PDATA : POINTER TO BYTE;
	BMOTOROLA : BOOL;
	PRESULT : POINTER TO UDINT;
END_VAR
END_METHOD

METHOD SWAP2 : IecVarAccess_Interfaces.XWORD
VAR_INPUT
	PDATA : POINTER TO BYTE;
	VARINFO : IecVarAccess_Interfaces.IVariableInformation;
	BMOTOROLA : BOOL;
	PRESULT : POINTER TO UDINT;
END_VAR
END_METHOD

(* ---- TYPEDESC_ALIAS.pou ---- *)
FUNCTION_BLOCK TYPEDESC_ALIAS EXTENDS TypeDesc
VAR
	_PSZNAME : POINTER TO STRING;
	_PIBASETYPEDESC : POINTER TO TypeDesc;
END_VAR
END_FUNCTION_BLOCK

METHOD FINDCHILD : ITreeWalker
VAR_INPUT
	PSTPATH : POINTER TO STRING;
	VARINFO : REFERENCE TO VariableInformation;
	PRESULT : POINTER TO UDINT;
END_VAR
VAR_IN_OUT
	IOFFSETINPATH : __XWORD;
END_VAR
END_METHOD

METHOD GETADDRESS : POINTER TO BYTE
VAR_INPUT
	PADDRESS : POINTER TO BYTE;
	PRESULT : POINTER TO UDINT;
END_VAR
END_METHOD

METHOD GETBASETYPE_INTERNAL : REFERENCE TO TypeDesc
END_METHOD

METHOD GETENUMVALUES_INTERNAL : POINTER TO EnumValues
VAR_INPUT
	PNNUMOFENUMVALUES : POINTER TO INT;
	PRESULT : POINTER TO RTS_IEC_RESULT;
END_VAR
END_METHOD

METHOD GETNAME_INTERNAL : POINTER TO STRING
VAR_INPUT
	PRESULT : POINTER TO SysTypes.RTS_IEC_RESULT;
END_VAR
END_METHOD

METHOD GETNATIVESIZE_INTERNAL : __XWORD
END_METHOD

METHOD GETSIZE2_INTERNAL : __XWORD
VAR_INPUT
	VARINFO : REFERENCE TO VariableInformation;
END_VAR
END_METHOD

METHOD GETSIZE_INTERNAL : __XWORD
END_METHOD

METHOD GETSWAPSIZE_INTERNAL : __XWORD
END_METHOD

METHOD GETTYPECLASS2_INTERNAL : TypeClass
VAR_INPUT
	DWFLAGS : DWORD;
END_VAR
END_METHOD

METHOD GETTYPECLASS_INTERNAL : TypeClass
END_METHOD

METHOD GETTYPEDESC_INTERNAL : UDINT
VAR_INPUT
	PTYPEDESCSTRUCT : POINTER TO TypeDescAsUnion;
END_VAR
END_METHOD

METHOD GETTYPENODE_INTERNAL : REFERENCE TO TypeDesc
VAR_INPUT
	VARINFO : REFERENCE TO VariableInformation;
	OPTIONS : WORD;
END_VAR
END_METHOD

METHOD GET_INTERNAL : __XWORD
VAR_INPUT
	PDEST : POINTER TO BYTE;
	PSRC : POINTER TO BYTE;
	VARINFO : REFERENCE TO VariableInformation;
	DWSIZE : __XWORD;
	PRESULT : POINTER TO UDINT;
END_VAR
END_METHOD

METHOD NODEFOUND_INTERNAL : UDINT
VAR_INPUT
	VARINFO : REFERENCE TO VariableInformation;
	BDIRECTCHILDFOUND : BOOL;
END_VAR
END_METHOD

METHOD SET_INTERNAL : __XWORD
VAR_INPUT
	PSRC : POINTER TO BYTE;
	PDEST : POINTER TO BYTE;
	VARINFO : REFERENCE TO VariableInformation;
	DWSIZE : __XWORD;
	PRESULT : POINTER TO UDINT;
END_VAR
END_METHOD

METHOD SWAP_INTERNAL : __XWORD
VAR_INPUT
	PDATA : POINTER TO BYTE;
	VARINFO : REFERENCE TO VariableInformation;
	DWSIZE : __XWORD;
	BMOTOROLA : BOOL;
	PRESULT : POINTER TO UDINT;
END_VAR
END_METHOD

(* ---- TYPEDESC_ALIASWITHATTRIBUTES.pou ---- *)
FUNCTION_BLOCK TYPEDESC_ALIASWITHATTRIBUTES EXTENDS TypeDesc_Alias
VAR
	_NUMOFATTRIBUTES : WORD;
	_PATTRIBUTES : POINTER TO ARRAY [0..0] OF POINTER TO STRING;
END_VAR
END_FUNCTION_BLOCK

METHOD GETATTRIBUTEBYINDEX_INTERNAL : POINTER TO STRING
VAR_INPUT
	WINDEX : WORD;
END_VAR
END_METHOD

METHOD GETENUMMEMBERATTRIBUTELIST_INTERNAL : POINTER TO EnumAttributes
VAR_INPUT
	PNNUMOFENUMVALUES : POINTER TO INT;
	PRESULT : POINTER TO RTS_IEC_RESULT;
END_VAR
END_METHOD

METHOD GETNUMOFATTRIBUTES_INTERNAL : WORD
END_METHOD

(* ---- TYPEDESC_ARRAY.pou ---- *)
FUNCTION_BLOCK TYPEDESC_ARRAY EXTENDS TypeDesc
VAR
	_DWNATIVESIZE : DWORD;
	_IDIMENSIONS : USINT;
	_DIMENSION : ARRAY [0..(MAX_ARRAY_DIMENSION - 1)] OF ArrayDimension;
	_IBASETYPEDESC : REFERENCE TO TypeDesc;
END_VAR
END_FUNCTION_BLOCK

METHOD BROWSEINTOTYPE : ITreeWalker
VAR_INPUT
	PNODE : ITreeWalker;
	PVARINFO : REFERENCE TO VariableInformation;
	PBROWSEINFO : POINTER TO RtsBrowseInfo;
END_VAR
END_METHOD

METHOD BROWSENEXTELEMENT : ITreeWalker
VAR_INPUT
	PNODE : ITreeWalker;
	PVARINFO : REFERENCE TO VariableInformation;
	PBROWSEINFO : POINTER TO RtsBrowseInfo;
END_VAR
END_METHOD

METHOD BROWSEOUTOFTYPE : ITreeWalker
VAR_INPUT
	PNODE : ITreeWalker;
	PVARINFO : REFERENCE TO VariableInformation;
	PBROWSEINFO : POINTER TO RtsBrowseInfo;
END_VAR
END_METHOD

METHOD FINDCHILD : ITreeWalker
VAR_INPUT
	PSTPATH : POINTER TO STRING;
	VARINFO : REFERENCE TO VariableInformation;
	PRESULT : POINTER TO UDINT;
END_VAR
VAR_IN_OUT
	IOFFSETINPATH : __XWORD;
END_VAR
END_METHOD

METHOD GETCLIENTSIDESIZEALIGNED : __XWORD
END_METHOD

METHOD GETELEMENTCOUNT : __XWORD
END_METHOD

METHOD GETNATIVESIZE2_INTERNAL : __XWORD
VAR_INPUT
	VARINFO : REFERENCE TO VariableInformation;
END_VAR
END_METHOD

METHOD GETNATIVESIZE_INTERNAL : __XWORD
END_METHOD

METHOD GETSIZE2_INTERNAL : __XWORD
VAR_INPUT
	VARINFO : REFERENCE TO VariableInformation;
END_VAR
END_METHOD

METHOD GETSIZE_INTERNAL : __XWORD
END_METHOD

METHOD GETTYPECLASS2_INTERNAL : TypeClass
VAR_INPUT
	DWFLAGS : DWORD;
END_VAR
END_METHOD

METHOD GETTYPECLASS_INTERNAL : TypeClass
END_METHOD

METHOD GETTYPEDESC_INTERNAL : UDINT
VAR_INPUT
	PTYPEDESCSTRUCT : POINTER TO TypeDescAsUnion;
END_VAR
END_METHOD

METHOD GETTYPENODE_INTERNAL : REFERENCE TO TypeDesc
VAR_INPUT
	VARINFO : REFERENCE TO VariableInformation;
	OPTIONS : WORD;
END_VAR
END_METHOD

METHOD GET_INTERNAL : __XWORD
VAR_INPUT
	PDEST : POINTER TO BYTE;
	PSRC : POINTER TO BYTE;
	VARINFO : REFERENCE TO VariableInformation;
	DWSIZE : __XWORD;
	PRESULT : POINTER TO UDINT;
END_VAR
END_METHOD

METHOD HANDLEBROWSEINFOANDOFFSET : RTS_IEC_RESULT
VAR_INPUT
	VARINFO : REFERENCE TO VariableInformation;
	PBROWSEINFO : POINTER TO RtsBrowseInfo;
	INDEX : DINT;
	OPERATION : BrowseOperation;
END_VAR
END_METHOD

METHOD NODEFOUND_INTERNAL : UDINT
VAR_INPUT
	VARINFO : REFERENCE TO VariableInformation;
	BDIRECTCHILDFOUND : BOOL;
END_VAR
END_METHOD

METHOD PARSEINDEX : RTS_IEC_RESULT
VAR_INPUT
	PSTPATH : POINTER TO STRING;
END_VAR
VAR_OUTPUT
	PARSEDINDEX : ARRAY [0..(MAX_ARRAY_DIMENSION - 1)] OF DINT;
	NUMPARSEDINDEX : INT;
	LENGHTFORNOTIFICATION : INT;
END_VAR
END_METHOD

METHOD SET_INTERNAL : __XWORD
VAR_INPUT
	PSRC : POINTER TO BYTE;
	PDEST : POINTER TO BYTE;
	VARINFO : REFERENCE TO VariableInformation;
	DWSIZE : __XWORD;
	PRESULT : POINTER TO UDINT;
END_VAR
END_METHOD

METHOD SWAP_INTERNAL : __XWORD
VAR_INPUT
	PDATA : POINTER TO BYTE;
	VARINFO : REFERENCE TO VariableInformation;
	DWSIZE : __XWORD;
	BMOTOROLA : BOOL;
	PRESULT : POINTER TO UDINT;
END_VAR
END_METHOD

METHOD USEARRAYBASETYPE : BOOL
VAR_INPUT
	VARINFO : REFERENCE TO VariableInformation;
END_VAR
END_METHOD

METHOD DECREMENTOFFSET
VAR_INPUT
	VARINFO : REFERENCE TO VariableInformation;
	ENTRIESCOUNT : DINT;
END_VAR
END_METHOD

METHOD INCREMENTOFFSET
VAR_INPUT
	VARINFO : REFERENCE TO VariableInformation;
	ENTRIESCOUNT : DINT;
END_VAR
END_METHOD

METHOD NOTIFYARRAYACCESS
VAR_INPUT
	PST : POINTER TO STRING;
	LEN : INT;
	VI : REFERENCE TO VariableInformation;
END_VAR
END_METHOD

METHOD PROTDONOTIFYARRAYACCESS
VAR_INPUT
	PST : POINTER TO STRING;
	LEN : INT;
	NOTFIYCLIENT : IArrayNotifiable;
END_VAR
END_METHOD

(* ---- TYPEDESC_ARRAY_BYTEADDRESSED.pou ---- *)
FUNCTION_BLOCK TYPEDESC_ARRAY_BYTEADDRESSED EXTENDS TypeDesc_Array
END_FUNCTION_BLOCK

METHOD GET_INTERNAL : __XWORD
VAR_INPUT
	PDEST : POINTER TO BYTE;
	PSRC : POINTER TO BYTE;
	VARINFO : REFERENCE TO VariableInformation;
	DWSIZE : __XWORD;
	PRESULT : POINTER TO UDINT;
END_VAR
END_METHOD

METHOD SET_INTERNAL : __XWORD
VAR_INPUT
	PSRC : POINTER TO BYTE;
	PDEST : POINTER TO BYTE;
	VARINFO : REFERENCE TO VariableInformation;
	DWSIZE : __XWORD;
	PRESULT : POINTER TO UDINT;
END_VAR
END_METHOD

METHOD INCREMENTOFFSET
VAR_INPUT
	VARINFO : REFERENCE TO VariableInformation;
	ENTRIESCOUNT : DINT;
END_VAR
END_METHOD

(* ---- TYPEDESC_ARRAY_REMOTE.pou ---- *)
FUNCTION_BLOCK TYPEDESC_ARRAY_REMOTE EXTENDS TypeDesc_Array
END_FUNCTION_BLOCK

METHOD INCREMENTOFFSET
VAR_INPUT
	VARINFO : REFERENCE TO VariableInformation;
	ENTRIESCOUNT : DINT;
END_VAR
END_METHOD

(* ---- TYPEDESC_ENUM.pou ---- *)
FUNCTION_BLOCK TYPEDESC_ENUM EXTENDS TypeDesc_Simple
VAR
	_PSZNAME : POINTER TO STRING;
	_NUMOFENUMVALUES : INT;
	_ENUMVALUES : POINTER TO ARRAY [0..0] OF EnumValues;
END_VAR
END_FUNCTION_BLOCK

METHOD GETENUMVALUES_INTERNAL : POINTER TO EnumValues
VAR_INPUT
	PNNUMOFENUMVALUES : POINTER TO INT;
	PRESULT : POINTER TO RTS_IEC_RESULT;
END_VAR
END_METHOD

METHOD GETNAME_INTERNAL : POINTER TO STRING
VAR_INPUT
	PRESULT : POINTER TO SysTypes.RTS_IEC_RESULT;
END_VAR
END_METHOD

METHOD GETTYPECLASS2_INTERNAL : TypeClass
VAR_INPUT
	DWFLAGS : DWORD;
END_VAR
END_METHOD

(* ---- TYPEDESC_ENUMWITHATTRIBUTES.pou ---- *)
FUNCTION_BLOCK TYPEDESC_ENUMWITHATTRIBUTES EXTENDS TypeDesc_Enum
VAR
	_NUMOFATTRIBUTES : WORD;
	_PATTRIBUTES : POINTER TO ARRAY [0..0] OF POINTER TO STRING;
	_PENUMATTRIBUTES : POINTER TO ARRAY [0..0] OF POINTER TO EnumAttributes;
END_VAR
END_FUNCTION_BLOCK

METHOD GETATTRIBUTEBYINDEX_INTERNAL : POINTER TO STRING
VAR_INPUT
	WINDEX : WORD;
END_VAR
END_METHOD

METHOD GETENUMMEMBERATTRIBUTELIST_INTERNAL : POINTER TO EnumAttributes
VAR_INPUT
	PNNUMOFENUMVALUES : POINTER TO INT;
	PRESULT : POINTER TO RTS_IEC_RESULT;
END_VAR
END_METHOD

METHOD GETNUMOFATTRIBUTES_INTERNAL : WORD
END_METHOD

(* ---- TYPEDESC_EXECUTABLE.pou ---- *)
FUNCTION_BLOCK TYPEDESC_EXECUTABLE EXTENDS TypeDesc_Struct2_WithBaseTypeAndAttributes
VAR
	_NMETHODCALLTYPEINDEX : WORD;
	_DEFININGSIGNATURE : REFERENCE TO TypeDesc;
	METHODCALLTYPEINDEX_INTERNAL : WORD;
END_VAR
END_FUNCTION_BLOCK

METHOD NODEFOUND_INTERNAL : UDINT
VAR_INPUT
	VARINFO : REFERENCE TO VariableInformation;
	BDIRECTCHILDFOUND : BOOL;
END_VAR
END_METHOD

(* ---- TYPEDESC_EXECUTABLE2.pou ---- *)
FUNCTION_BLOCK TYPEDESC_EXECUTABLE2 EXTENDS TypeDesc_Struct2_WithBaseTypeAndAttributes
VAR
	_METHODADR : POINTER TO POINTER TO BYTE;
	_SETINSTANCEPOINTER : BOOL;
	_DEFININGSIGNATURE : REFERENCE TO TypeDesc;
END_VAR
END_FUNCTION_BLOCK

METHOD EXECUTE_INTERNAL : RTS_IEC_RESULT
VAR_INPUT
	VARINFO : REFERENCE TO VariableInformation;
	PINST : POINTER TO BYTE;
	PMETHODPARAMS : POINTER TO BYTE;
	METHODPRAMSSIZE : __XWORD;
END_VAR
END_METHOD

METHOD GETMETHODARGUMENTS : SysTypes.RTS_IEC_RESULT
VAR_OUTPUT
	PINPUTARGUMENTS : POINTER TO CmpOPCUAStack_Interfaces.OpcUa_NodeId;
	POUTPUTARGUMENTS : POINTER TO CmpOPCUAStack_Interfaces.OpcUa_NodeId;
END_VAR
END_METHOD

METHOD NODEFOUND_INTERNAL : UDINT
VAR_INPUT
	VARINFO : REFERENCE TO VariableInformation;
	BDIRECTCHILDFOUND : BOOL;
END_VAR
END_METHOD

(* ---- TYPEDESC_OPCUABUILTINTYPE.pou ---- *)
FUNCTION_BLOCK TYPEDESC_OPCUABUILTINTYPE EXTENDS TypeDesc
VAR
	_BUILTINTYPE : OpcUa_BuiltInType;
	_SIZES : ARRAY [0..25] OF __XWORD := [0, SIZEOF(OpcUa_Boolean), SIZEOF(OpcUa_SByte), SIZEOF(OpcUa_Byte), SIZEOF(OpcUa_Int16), SIZEOF(OpcUa_UInt16), SIZEOF(OpcUa_Int32), SIZEOF(OpcUa_UInt32), SIZEOF(OpcUa_Int64), SIZEOF(OpcUa_UInt64), SIZEOF(OpcUa_Float), SIZEOF(OpcUa_Double), SIZEOF(OpcUa_String), SIZEOF(OpcUa_DateTime), SIZEOF(OpcUa_Guid), SIZEOF(OpcUa_ByteString), SIZEOF(OpcUa_ByteString), SIZEOF(OpcUa_NodeId), SIZEOF(OpcUa_ExpandedNodeId), SIZEOF(OpcUa_StatusCode), SIZEOF(OpcUa_QualifiedName), SIZEOF(OpcUa_LocalizedText), SIZEOF(OpcUa_ExtensionObject), SIZEOF(OpcUa_DataValue), SIZEOF(OpcUa_Variant), SIZEOF(OpcUa_DiagnosticInfo)];
END_VAR
END_FUNCTION_BLOCK

METHOD FINDCHILD : ITreeWalker
VAR_INPUT
	PSTPATH : POINTER TO STRING;
	VARINFO : REFERENCE TO VariableInformation;
	PRESULT : POINTER TO UDINT;
END_VAR
VAR_IN_OUT
	IOFFSETINPATH : __XWORD;
END_VAR
END_METHOD

METHOD GETNATIVESIZE2_INTERNAL : __XWORD
VAR_INPUT
	VARINFO : REFERENCE TO VariableInformation;
END_VAR
END_METHOD

METHOD GETNATIVESIZE_INTERNAL : __XWORD
END_METHOD

METHOD GETSIZE2_INTERNAL : __XWORD
VAR_INPUT
	VARINFO : REFERENCE TO VariableInformation;
END_VAR
END_METHOD

METHOD GETSIZE_INTERNAL : __XWORD
END_METHOD

METHOD GETTYPECLASS2_INTERNAL : TypeClass
VAR_INPUT
	DWFLAGS : DWORD;
END_VAR
END_METHOD

METHOD GETTYPECLASS_INTERNAL : TypeClass
END_METHOD

METHOD GETTYPEDESC_INTERNAL : UDINT
VAR_INPUT
	PTYPEDESCSTRUCT : POINTER TO TypeDescAsUnion;
END_VAR
END_METHOD

METHOD GETUABUILTINTYPE_INTERNAL : OpcUa_BuiltInType
END_METHOD

METHOD GET_INTERNAL : __XWORD
VAR_INPUT
	PDEST : POINTER TO BYTE;
	PSRC : POINTER TO BYTE;
	VARINFO : REFERENCE TO VariableInformation;
	DWSIZE : __XWORD;
	PRESULT : POINTER TO UDINT;
END_VAR
END_METHOD

METHOD NODEFOUND_INTERNAL : UDINT
VAR_INPUT
	VARINFO : REFERENCE TO VariableInformation;
	BDIRECTCHILDFOUND : BOOL;
END_VAR
END_METHOD

METHOD SET_INTERNAL : __XWORD
VAR_INPUT
	PSRC : POINTER TO BYTE;
	PDEST : POINTER TO BYTE;
	VARINFO : REFERENCE TO VariableInformation;
	DWSIZE : __XWORD;
	PRESULT : POINTER TO UDINT;
END_VAR
END_METHOD

METHOD SWAP_INTERNAL : __XWORD
VAR_INPUT
	PDATA : POINTER TO BYTE;
	VARINFO : REFERENCE TO VariableInformation;
	DWSIZE : __XWORD;
	BMOTOROLA : BOOL;
	PRESULT : POINTER TO UDINT;
END_VAR
END_METHOD

(* ---- TYPEDESC_PROPERTY.pou ---- *)
FUNCTION_BLOCK TYPEDESC_PROPERTY EXTENDS TypeDesc
VAR
	_IBASETYPEDESC : REFERENCE TO TypeDesc;
	_TYPECLASS : TypeClass;
	_MAXNESTINGDEPTH : UINT;
END_VAR
END_FUNCTION_BLOCK

METHOD BROWSEINTOTYPE : ITreeWalker
VAR_INPUT
	PNODE : ITreeWalker;
	PVARINFO : REFERENCE TO VariableInformation;
	PBROWSEINFO : POINTER TO RtsBrowseInfo;
END_VAR
END_METHOD

METHOD BROWSEOUTOFTYPE : ITreeWalker
VAR_INPUT
	PNODE : ITreeWalker;
	PVARINFO : REFERENCE TO VariableInformation;
	PBROWSEINFO : POINTER TO RtsBrowseInfo;
END_VAR
END_METHOD

METHOD FINDCHILD : ITreeWalker
VAR_INPUT
	PSTPATH : POINTER TO STRING;
	VARINFO : REFERENCE TO VariableInformation;
	PRESULT : POINTER TO UDINT;
END_VAR
VAR_IN_OUT
	IOFFSETINPATH : __XWORD;
END_VAR
END_METHOD

METHOD GETATTRIBUTEBYINDEX_INTERNAL : POINTER TO STRING
VAR_INPUT
	WINDEX : WORD;
END_VAR
END_METHOD

METHOD GETBASETYPE_INTERNAL : REFERENCE TO TypeDesc
END_METHOD

METHOD GETENUMMEMBERATTRIBUTELIST_INTERNAL : POINTER TO EnumAttributes
VAR_INPUT
	PNNUMOFENUMVALUES : POINTER TO INT;
	PRESULT : POINTER TO RTS_IEC_RESULT;
END_VAR
END_METHOD

METHOD GETENUMVALUES_INTERNAL : POINTER TO EnumValues
VAR_INPUT
	PNNUMOFENUMVALUES : POINTER TO INT;
	PRESULT : POINTER TO RTS_IEC_RESULT;
END_VAR
END_METHOD

METHOD GETNAME_INTERNAL : POINTER TO STRING
VAR_INPUT
	PRESULT : POINTER TO SysTypes.RTS_IEC_RESULT;
END_VAR
END_METHOD

METHOD GETNATIVESIZE2_INTERNAL : __XWORD
VAR_INPUT
	VARINFO : REFERENCE TO VariableInformation;
END_VAR
END_METHOD

METHOD GETNATIVESIZE_INTERNAL : __XWORD
END_METHOD

METHOD GETNUMOFATTRIBUTES_INTERNAL : WORD
END_METHOD

METHOD GETSIZE2_INTERNAL : __XWORD
VAR_INPUT
	VARINFO : REFERENCE TO VariableInformation;
END_VAR
END_METHOD

METHOD GETSIZE_INTERNAL : __XWORD
END_METHOD

METHOD GETSWAPSIZE_INTERNAL : __XWORD
END_METHOD

METHOD GETTYPECLASS2_INTERNAL : TypeClass
VAR_INPUT
	DWFLAGS : DWORD;
END_VAR
END_METHOD

METHOD GETTYPECLASS_INTERNAL : TypeClass
END_METHOD

METHOD GETTYPEDESC_INTERNAL : UDINT
VAR_INPUT
	PTYPEDESCSTRUCT : POINTER TO TypeDescAsUnion;
END_VAR
END_METHOD

METHOD GETTYPENODE_INTERNAL : REFERENCE TO TypeDesc
VAR_INPUT
	VARINFO : REFERENCE TO VariableInformation;
	OPTIONS : WORD;
END_VAR
END_METHOD

METHOD GET_INTERNAL : __XWORD
VAR_INPUT
	PDEST : POINTER TO BYTE;
	PSRC : POINTER TO BYTE;
	VARINFO : REFERENCE TO VariableInformation;
	DWSIZE : __XWORD;
	PRESULT : POINTER TO UDINT;
END_VAR
END_METHOD

METHOD HANDLEVARINFO : RTS_IEC_RESULT
VAR_INPUT
	VARINFO : REFERENCE TO VariableInformation;
	OPERATION : BrowseOperation;
END_VAR
END_METHOD

METHOD ISMEMBER : BOOL
VAR_INPUT
	PNODE : ITreeWalker;
END_VAR
END_METHOD

METHOD NODEFOUND_INTERNAL : UDINT
VAR_INPUT
	VARINFO : REFERENCE TO VariableInformation;
	BDIRECTCHILDFOUND : BOOL;
END_VAR
END_METHOD

METHOD SET_INTERNAL : __XWORD
VAR_INPUT
	PSRC : POINTER TO BYTE;
	PDEST : POINTER TO BYTE;
	VARINFO : REFERENCE TO VariableInformation;
	DWSIZE : __XWORD;
	PRESULT : POINTER TO UDINT;
END_VAR
END_METHOD

METHOD SWAP_INTERNAL : __XWORD
VAR_INPUT
	PDATA : POINTER TO BYTE;
	VARINFO : REFERENCE TO VariableInformation;
	DWSIZE : __XWORD;
	BMOTOROLA : BOOL;
	PRESULT : POINTER TO UDINT;
END_VAR
END_METHOD

(* ---- TYPEDESC_PROPERTY_REMOTE.pou ---- *)
FUNCTION_BLOCK TYPEDESC_PROPERTY_REMOTE EXTENDS TypeDesc_simple
VAR
	_IBASETYPEDESC : REFERENCE TO TypeDesc;
	_INFO : PropertyInfoRemote;
END_VAR
END_FUNCTION_BLOCK

METHOD GETBASETYPE_INTERNAL : REFERENCE TO TypeDesc
END_METHOD

METHOD GETTYPECLASS2_INTERNAL : TypeClass
VAR_INPUT
	DWFLAGS : DWORD;
END_VAR
END_METHOD

METHOD GET_INTERNAL : __XWORD
VAR_INPUT
	PDEST : POINTER TO BYTE;
	PSRC : POINTER TO BYTE;
	VARINFO : REFERENCE TO VariableInformation;
	DWSIZE : __XWORD;
	PRESULT : POINTER TO UDINT;
END_VAR
END_METHOD

METHOD SET_INTERNAL : __XWORD
VAR_INPUT
	PSRC : POINTER TO BYTE;
	PDEST : POINTER TO BYTE;
	VARINFO : REFERENCE TO VariableInformation;
	DWSIZE : __XWORD;
	PRESULT : POINTER TO UDINT;
END_VAR
END_METHOD

(* ---- TYPEDESC_REFERENCE.pou ---- *)
FUNCTION_BLOCK TYPEDESC_REFERENCE EXTENDS TypeDesc
VAR
	_IBASETYPEDESC : REFERENCE TO TypeDesc;
	_TYPECLASS : TypeClass;
	_DWSWAPSIZE : DWORD;
	_MAXNESTINGDEPTH : UINT;
	_PSZNAME : POINTER TO STRING;
END_VAR
END_FUNCTION_BLOCK

METHOD BROWSEINTOTYPE : ITreeWalker
VAR_INPUT
	PNODE : ITreeWalker;
	PVARINFO : REFERENCE TO VariableInformation;
	PBROWSEINFO : POINTER TO RtsBrowseInfo;
END_VAR
END_METHOD

METHOD BROWSEOUTOFTYPE : ITreeWalker
VAR_INPUT
	PNODE : ITreeWalker;
	PVARINFO : REFERENCE TO VariableInformation;
	PBROWSEINFO : POINTER TO RtsBrowseInfo;
END_VAR
END_METHOD

METHOD CALCULATEADDRESS : REFERENCE TO TypeDesc
VAR_INPUT
	BASEADDRESS : __XWORD;
	VARINFO : REFERENCE TO VariableInformation;
END_VAR
VAR_OUTPUT
	RESULT : RTS_IEC_RESULT;
	ADDRESS : __XWORD;
	TARGETNODE : ILeafTreeNode;
END_VAR
END_METHOD

METHOD DEREFERENCE : REFERENCE TO TypeDesc
VAR_INPUT
	VARINFO : REFERENCE TO VariableInformation;
	PIECADRESS : POINTER TO BYTE;
	UPDATEADRESSINVARINFO : BOOL;
END_VAR
VAR_OUTPUT
	TARGETNODE : ILeafTreeNode;
	PADDRESS : POINTER TO BYTE;
	RESULT : RTS_IEC_RESULT;
END_VAR
END_METHOD

METHOD FINDCHILD : ITreeWalker
VAR_INPUT
	PSTPATH : POINTER TO STRING;
	VARINFO : REFERENCE TO VariableInformation;
	PRESULT : POINTER TO UDINT;
END_VAR
VAR_IN_OUT
	IOFFSETINPATH : __XWORD;
END_VAR
END_METHOD

METHOD GETATTRIBUTEBYINDEX_INTERNAL : POINTER TO STRING
VAR_INPUT
	WINDEX : WORD;
END_VAR
END_METHOD

METHOD GETBASETYPE_INTERNAL : REFERENCE TO TypeDesc
END_METHOD

METHOD GETENUMMEMBERATTRIBUTELIST_INTERNAL : POINTER TO EnumAttributes
VAR_INPUT
	PNNUMOFENUMVALUES : POINTER TO INT;
	PRESULT : POINTER TO RTS_IEC_RESULT;
END_VAR
END_METHOD

METHOD GETENUMVALUES_INTERNAL : POINTER TO EnumValues
VAR_INPUT
	PNNUMOFENUMVALUES : POINTER TO INT;
	PRESULT : POINTER TO RTS_IEC_RESULT;
END_VAR
END_METHOD

METHOD GETNAME_INTERNAL : POINTER TO STRING
VAR_INPUT
	PRESULT : POINTER TO SysTypes.RTS_IEC_RESULT;
END_VAR
END_METHOD

METHOD GETNATIVESIZE2_INTERNAL : __XWORD
VAR_INPUT
	VARINFO : REFERENCE TO VariableInformation;
END_VAR
END_METHOD

METHOD GETNATIVESIZE_INTERNAL : __XWORD
END_METHOD

METHOD GETNUMOFATTRIBUTES_INTERNAL : WORD
END_METHOD

METHOD GETREFERENCEBASETYPE_INTERNAL : REFERENCE TO TypeDesc
VAR_INPUT
	PRESULT : POINTER TO RTS_IEC_RESULT;
END_VAR
END_METHOD

METHOD GETSIZE2_INTERNAL : __XWORD
VAR_INPUT
	VARINFO : REFERENCE TO VariableInformation;
END_VAR
END_METHOD

METHOD GETSIZE_INTERNAL : __XWORD
END_METHOD

METHOD GETSWAPSIZE_INTERNAL : __XWORD
END_METHOD

METHOD GETTYPECLASS2_INTERNAL : TypeClass
VAR_INPUT
	DWFLAGS : DWORD;
END_VAR
END_METHOD

METHOD GETTYPECLASS_INTERNAL : TypeClass
END_METHOD

METHOD GETTYPEDESC_INTERNAL : UDINT
VAR_INPUT
	PTYPEDESCSTRUCT : POINTER TO TypeDescAsUnion;
END_VAR
END_METHOD

METHOD GETTYPENODE_INTERNAL : REFERENCE TO TypeDesc
VAR_INPUT
	VARINFO : REFERENCE TO VariableInformation;
	OPTIONS : WORD;
END_VAR
END_METHOD

METHOD GET_INTERNAL : __XWORD
VAR_INPUT
	PDEST : POINTER TO BYTE;
	PSRC : POINTER TO BYTE;
	VARINFO : REFERENCE TO VariableInformation;
	DWSIZE : __XWORD;
	PRESULT : POINTER TO UDINT;
END_VAR
END_METHOD

METHOD HANDLEVARINFO : RTS_IEC_RESULT
VAR_INPUT
	VARINFO : REFERENCE TO VariableInformation;
	OPERATION : BrowseOperation;
END_VAR
END_METHOD

METHOD ISMEMBER : BOOL
VAR_INPUT
	PNODE : ITreeWalker;
END_VAR
END_METHOD

METHOD NODEFOUND_INTERNAL : UDINT
VAR_INPUT
	VARINFO : REFERENCE TO VariableInformation;
	BDIRECTCHILDFOUND : BOOL;
END_VAR
END_METHOD

METHOD SET_INTERNAL : __XWORD
VAR_INPUT
	PSRC : POINTER TO BYTE;
	PDEST : POINTER TO BYTE;
	VARINFO : REFERENCE TO VariableInformation;
	DWSIZE : __XWORD;
	PRESULT : POINTER TO UDINT;
END_VAR
END_METHOD

METHOD SWAP_INTERNAL : __XWORD
VAR_INPUT
	PDATA : POINTER TO BYTE;
	VARINFO : REFERENCE TO VariableInformation;
	DWSIZE : __XWORD;
	BMOTOROLA : BOOL;
	PRESULT : POINTER TO UDINT;
END_VAR
END_METHOD

(* ---- TYPEDESC_SIMPLE.pou ---- *)
FUNCTION_BLOCK TYPEDESC_SIMPLE EXTENDS TypeDesc
VAR
	_TYPECLASS : TypeClass;
	_DWSWAPSIZE : DWORD;
END_VAR
END_FUNCTION_BLOCK

METHOD FINDCHILD : ITreeWalker
VAR_INPUT
	PSTPATH : POINTER TO STRING;
	VARINFO : REFERENCE TO VariableInformation;
	PRESULT : POINTER TO UDINT;
END_VAR
VAR_IN_OUT
	IOFFSETINPATH : __XWORD;
END_VAR
END_METHOD

METHOD GETSWAPSIZE_INTERNAL : __XWORD
END_METHOD

METHOD GETTYPECLASS_INTERNAL : TypeClass
END_METHOD

METHOD GETTYPEDESC_INTERNAL : UDINT
VAR_INPUT
	PTYPEDESCSTRUCT : POINTER TO TypeDescAsUnion;
END_VAR
END_METHOD

METHOD GET_INTERNAL : __XWORD
VAR_INPUT
	PDEST : POINTER TO BYTE;
	PSRC : POINTER TO BYTE;
	VARINFO : REFERENCE TO VariableInformation;
	DWSIZE : __XWORD;
	PRESULT : POINTER TO UDINT;
END_VAR
END_METHOD

METHOD NODEFOUND_INTERNAL : UDINT
VAR_INPUT
	VARINFO : REFERENCE TO VariableInformation;
	BDIRECTCHILDFOUND : BOOL;
END_VAR
END_METHOD

METHOD SET_INTERNAL : __XWORD
VAR_INPUT
	PSRC : POINTER TO BYTE;
	PDEST : POINTER TO BYTE;
	VARINFO : REFERENCE TO VariableInformation;
	DWSIZE : __XWORD;
	PRESULT : POINTER TO UDINT;
END_VAR
END_METHOD

METHOD SWAP_INTERNAL : __XWORD
VAR_INPUT
	PDATA : POINTER TO BYTE;
	VARINFO : REFERENCE TO VariableInformation;
	DWSIZE : __XWORD;
	BMOTOROLA : BOOL;
	PRESULT : POINTER TO UDINT;
END_VAR
END_METHOD

(* ---- TYPEDESC_SIMPLE_BIT.pou ---- *)
FUNCTION_BLOCK TYPEDESC_SIMPLE_BIT EXTENDS TypeDesc_Simple
VAR
	_BYBITOFFSET : BYTE;
END_VAR
END_FUNCTION_BLOCK

METHOD GET_INTERNAL : __XWORD
VAR_INPUT
	PDEST : POINTER TO BYTE;
	PSRC : POINTER TO BYTE;
	VARINFO : REFERENCE TO VariableInformation;
	DWSIZE : __XWORD;
	PRESULT : POINTER TO UDINT;
END_VAR
END_METHOD

METHOD NODEFOUND_INTERNAL : UDINT
VAR_INPUT
	VARINFO : REFERENCE TO VariableInformation;
	BDIRECTCHILDFOUND : BOOL;
END_VAR
END_METHOD

METHOD SET_INTERNAL : __XWORD
VAR_INPUT
	PSRC : POINTER TO BYTE;
	PDEST : POINTER TO BYTE;
	VARINFO : REFERENCE TO VariableInformation;
	DWSIZE : __XWORD;
	PRESULT : POINTER TO UDINT;
END_VAR
END_METHOD

(* ---- TYPEDESC_STRUCT.pou ---- *)
FUNCTION_BLOCK TYPEDESC_STRUCT EXTENDS TypeDesc
VAR
	_DWNATIVESIZE : DWORD;
	_ICOMPONENTS : DINT;
	_COMPONENTS : POINTER TO ARRAY [0..0] OF POINTER TO LeafTreeNode;
	_SORTEDCOMPONENTS : POINTER TO ARRAY [0..0] OF POINTER TO LeafTreeNode;
	_SORTEDBYBROWSENAME : POINTER TO POINTER TO SymbolsBaseNode;
END_VAR
END_FUNCTION_BLOCK

METHOD BROWSEINTOTYPE : ITreeWalker
VAR_INPUT
	PNODE : ITreeWalker;
	PVARINFO : REFERENCE TO VariableInformation;
	PBROWSEINFO : POINTER TO RtsBrowseInfo;
END_VAR
END_METHOD

METHOD BROWSENEXTELEMENT : ITreeWalker
VAR_INPUT
	PNODE : ITreeWalker;
	PVARINFO : REFERENCE TO VariableInformation;
	PBROWSEINFO : POINTER TO RtsBrowseInfo;
END_VAR
END_METHOD

METHOD BROWSEOUTOFTYPE : ITreeWalker
VAR_INPUT
	PNODE : ITreeWalker;
	PVARINFO : REFERENCE TO VariableInformation;
	PBROWSEINFO : POINTER TO RtsBrowseInfo;
END_VAR
END_METHOD

METHOD FINDCHILD : ITreeWalker
VAR_INPUT
	PSTPATH : POINTER TO STRING;
	VARINFO : REFERENCE TO VariableInformation;
	PRESULT : POINTER TO UDINT;
END_VAR
VAR_IN_OUT
	IOFFSETINPATH : __XWORD;
END_VAR
END_METHOD

METHOD GETNATIVESIZE_INTERNAL : __XWORD
END_METHOD

METHOD GETTYPECLASS_INTERNAL : TypeClass
END_METHOD

METHOD GETTYPEDESC_INTERNAL : UDINT
VAR_INPUT
	PTYPEDESCSTRUCT : POINTER TO TypeDescAsUnion;
END_VAR
END_METHOD

METHOD GET_INTERNAL : __XWORD
VAR_INPUT
	PDEST : POINTER TO BYTE;
	PSRC : POINTER TO BYTE;
	VARINFO : REFERENCE TO VariableInformation;
	DWSIZE : __XWORD;
	PRESULT : POINTER TO UDINT;
END_VAR
END_METHOD

METHOD HANDLEBROWSEINFOANDOFFSET : RTS_IEC_RESULT
VAR_INPUT
	PNODE : POINTER TO LeafTreeNode;
	VARINFO : REFERENCE TO VariableInformation;
	PBROWSEINFO : POINTER TO RtsBrowseInfo;
	INDEX : DINT;
	OPERATION : BrowseOperation;
END_VAR
END_METHOD

METHOD HANDLEFOUNDCHILD : RTS_IEC_RESULT
VAR_INPUT
	PNODE : POINTER TO LeafTreeNode;
	VARINFO : REFERENCE TO VariableInformation;
END_VAR
END_METHOD

METHOD ISMEMBER : BOOL
VAR_INPUT
	PNODE : ITreeWalker;
END_VAR
END_METHOD

METHOD NODEFOUND_INTERNAL : UDINT
VAR_INPUT
	VARINFO : REFERENCE TO VariableInformation;
	BDIRECTCHILDFOUND : BOOL;
END_VAR
END_METHOD

METHOD SEARCHMEMBER : POINTER TO LeafTreeNode
VAR_INPUT
	NAME : POINTER TO STRING;
	NAMELEN : DINT;
	PRESULT : POINTER TO RTS_IEC_RESULT;
END_VAR
VAR_OUTPUT
	INDEX : DINT;
END_VAR
END_METHOD

METHOD SET_INTERNAL : __XWORD
VAR_INPUT
	PSRC : POINTER TO BYTE;
	PDEST : POINTER TO BYTE;
	VARINFO : REFERENCE TO VariableInformation;
	DWSIZE : __XWORD;
	PRESULT : POINTER TO UDINT;
END_VAR
END_METHOD

METHOD SWAP_INTERNAL : __XWORD
VAR_INPUT
	PDATA : POINTER TO BYTE;
	VARINFO : REFERENCE TO VariableInformation;
	DWSIZE : __XWORD;
	BMOTOROLA : BOOL;
	PRESULT : POINTER TO UDINT;
END_VAR
END_METHOD

METHOD GETFIRSTCHILDBYBROWSENAME : ITreeWalker
VAR_INPUT
	PBROWSENAME : POINTER TO OpcUa_QualifiedName;
	VARINFO : REFERENCE TO VariableInformation;
END_VAR
VAR_OUTPUT
	RESULT : RTS_IEC_RESULT;
END_VAR
END_METHOD

METHOD GETNEXTCHILDBYBROWSENAME : ITreeWalker
VAR_INPUT
	PBROWSENAME : POINTER TO OpcUa_QualifiedName;
	VARINFO : REFERENCE TO VariableInformation;
	PBROWSEINFO : POINTER TO RtsBrowseInfo;
END_VAR
VAR_OUTPUT
	RESULT : RTS_IEC_RESULT;
END_VAR
END_METHOD

METHOD PROTTOKENLENGTH : DINT
VAR_INPUT
	PST : POINTER TO STRING;
END_VAR
END_METHOD

(* ---- TYPEDESC_STRUCT2.pou ---- *)
FUNCTION_BLOCK TYPEDESC_STRUCT2 EXTENDS TypeDesc_Struct
VAR
	_PSZNAME : POINTER TO STRING;
	_TYPECLASS : TypeClass := TypeClass.TYPE_USERDEF;
END_VAR
END_FUNCTION_BLOCK

METHOD GETNAME_INTERNAL : POINTER TO STRING
VAR_INPUT
	PRESULT : POINTER TO SysTypes.RTS_IEC_RESULT;
END_VAR
END_METHOD

METHOD GETTYPECLASS2_INTERNAL : TypeClass
VAR_INPUT
	DWFLAGS : DWORD;
END_VAR
END_METHOD

(* ---- TYPEDESC_STRUCT2_WITHBASETYPE.pou ---- *)
FUNCTION_BLOCK TYPEDESC_STRUCT2_WITHBASETYPE EXTENDS TypeDesc_Struct2
VAR
	_IBASETYPEDESC : REFERENCE TO TypeDesc;
END_VAR
END_FUNCTION_BLOCK

METHOD GETBASETYPE_INTERNAL : REFERENCE TO TypeDesc
END_METHOD

METHOD GETTYPECLASS2_INTERNAL : TypeClass
VAR_INPUT
	DWFLAGS : DWORD;
END_VAR
END_METHOD

(* ---- TYPEDESC_STRUCT2_WITHBASETYPEANDATTRIBUTES.pou ---- *)
FUNCTION_BLOCK TYPEDESC_STRUCT2_WITHBASETYPEANDATTRIBUTES EXTENDS TypeDesc_Struct2_WithBaseType
VAR
	_NUMOFATTRIBUTES : WORD;
	_PATTRIBUTES : POINTER TO ARRAY [0..0] OF POINTER TO STRING;
END_VAR
END_FUNCTION_BLOCK

METHOD GETATTRIBUTEBYINDEX_INTERNAL : POINTER TO STRING
VAR_INPUT
	WINDEX : WORD;
END_VAR
END_METHOD

METHOD GETENUMMEMBERATTRIBUTELIST_INTERNAL : POINTER TO EnumAttributes
VAR_INPUT
	PNNUMOFENUMVALUES : POINTER TO INT;
	PRESULT : POINTER TO RTS_IEC_RESULT;
END_VAR
END_METHOD

METHOD GETNUMOFATTRIBUTES_INTERNAL : WORD
END_METHOD

(* ---- TYPEDESC_STRUCT_DERIVED_REMOTE.pou ---- *)
FUNCTION_BLOCK TYPEDESC_STRUCT_DERIVED_REMOTE EXTENDS TypeDesc_Struct_Remote
VAR
	_IBASETYPEDESC : REFERENCE TO TypeDesc;
END_VAR
END_FUNCTION_BLOCK

METHOD FINDCHILD : ITreeWalker
VAR_INPUT
	PSTPATH : POINTER TO STRING;
	VARINFO : REFERENCE TO VariableInformation;
	PRESULT : POINTER TO UDINT;
END_VAR
VAR_IN_OUT
	IOFFSETINPATH : __XWORD;
END_VAR
END_METHOD

(* ---- TYPEDESC_STRUCT_REMOTE.pou ---- *)
FUNCTION_BLOCK TYPEDESC_STRUCT_REMOTE EXTENDS TypeDesc_Struct
VAR
	_DWLOCALNATIVESIZE : DWORD;
END_VAR
END_FUNCTION_BLOCK

METHOD GETSECONDNATIVESIZE : DWORD
END_METHOD

(* ---- TYPEDESC_SUBRANGE.pou ---- *)
FUNCTION_BLOCK TYPEDESC_SUBRANGE EXTENDS TypeDesc_Simple
VAR
	_PSZNAME : POINTER TO STRING;
	_IBASETYPEDESC : REFERENCE TO TypeDesc;
	_LWLOWERBORDER : LWORD;
	_LWUPPERBORDER : LWORD;
END_VAR
END_FUNCTION_BLOCK

METHOD GETBASETYPE_INTERNAL : REFERENCE TO TypeDesc
END_METHOD

METHOD GETNAME_INTERNAL : POINTER TO STRING
VAR_INPUT
	PRESULT : POINTER TO SysTypes.RTS_IEC_RESULT;
END_VAR
END_METHOD

METHOD GETRANGE_INTERNAL : BOOL
VAR_INPUT
	PLOWER : POINTER TO LWORD;
	PUPPER : POINTER TO LWORD;
END_VAR
END_METHOD

METHOD GETTYPECLASS2_INTERNAL : TypeClass
VAR_INPUT
	DWFLAGS : DWORD;
END_VAR
END_METHOD

METHOD GET_INTERNAL : __XWORD
VAR_INPUT
	PDEST : POINTER TO BYTE;
	PSRC : POINTER TO BYTE;
	VARINFO : REFERENCE TO VariableInformation;
	DWSIZE : __XWORD;
	PRESULT : POINTER TO UDINT;
END_VAR
END_METHOD

METHOD SET_INTERNAL : __XWORD
VAR_INPUT
	PSRC : POINTER TO BYTE;
	PDEST : POINTER TO BYTE;
	VARINFO : REFERENCE TO VariableInformation;
	DWSIZE : __XWORD;
	PRESULT : POINTER TO UDINT;
END_VAR
END_METHOD

(* ---- TYPEDESC_UAPROPERTIES.pou ---- *)
FUNCTION_BLOCK TYPEDESC_UAPROPERTIES EXTENDS TypeDesc_Struct
VAR
	BASETYPEDESC : REFERENCE TO TypeDesc;
	OFFSET : __XWORD;
	METHODCALLTYPEINDEX_INTERNAL : WORD;
END_VAR
END_FUNCTION_BLOCK

METHOD BROWSEINTOTYPE : ITreeWalker
VAR_INPUT
	PNODE : ITreeWalker;
	PVARINFO : REFERENCE TO VariableInformation;
	PBROWSEINFO : POINTER TO RtsBrowseInfo;
END_VAR
END_METHOD

METHOD BROWSENEXTELEMENT : ITreeWalker
VAR_INPUT
	PNODE : ITreeWalker;
	PVARINFO : REFERENCE TO VariableInformation;
	PBROWSEINFO : POINTER TO RtsBrowseInfo;
END_VAR
END_METHOD

METHOD FINDCHILD : ITreeWalker
VAR_INPUT
	PSTPATH : POINTER TO STRING;
	VARINFO : REFERENCE TO VariableInformation;
	PRESULT : POINTER TO UDINT;
END_VAR
VAR_IN_OUT
	IOFFSETINPATH : __XWORD;
END_VAR
END_METHOD

METHOD GETFIRSTCHILDBYBROWSENAME : ITreeWalker
VAR_INPUT
	PBROWSENAME : POINTER TO OpcUa_QualifiedName;
	VARINFO : REFERENCE TO VariableInformation;
END_VAR
VAR_OUTPUT
	RESULT : RTS_IEC_RESULT;
END_VAR
END_METHOD

METHOD GETNEXTCHILDBYBROWSENAME : ITreeWalker
VAR_INPUT
	PBROWSENAME : POINTER TO OpcUa_QualifiedName;
	VARINFO : REFERENCE TO VariableInformation;
	PBROWSEINFO : POINTER TO RtsBrowseInfo;
END_VAR
VAR_OUTPUT
	RESULT : RTS_IEC_RESULT;
END_VAR
END_METHOD

METHOD GET_INTERNAL : __XWORD
VAR_INPUT
	PDEST : POINTER TO BYTE;
	PSRC : POINTER TO BYTE;
	VARINFO : REFERENCE TO VariableInformation;
	DWSIZE : __XWORD;
	PRESULT : POINTER TO UDINT;
END_VAR
END_METHOD

METHOD ISMEMBER : BOOL
VAR_INPUT
	PNODE : ITreeWalker;
END_VAR
END_METHOD

METHOD SET_INTERNAL : __XWORD
VAR_INPUT
	PSRC : POINTER TO BYTE;
	PDEST : POINTER TO BYTE;
	VARINFO : REFERENCE TO VariableInformation;
	DWSIZE : __XWORD;
	PRESULT : POINTER TO UDINT;
END_VAR
END_METHOD

METHOD EXECUTE_INTERNAL : RTS_IEC_RESULT
VAR_INPUT
	VARINFO : REFERENCE TO VariableInformation;
	PINST : POINTER TO BYTE;
	PMETHODPARAMS : POINTER TO BYTE;
	METHODPRAMSSIZE : __XWORD;
END_VAR
END_METHOD

METHOD GETADDRESS : POINTER TO BYTE
VAR_INPUT
	PADDRESS : POINTER TO BYTE;
	PRESULT : POINTER TO UDINT;
END_VAR
END_METHOD

METHOD GETATTRIBUTEBYINDEX_INTERNAL : POINTER TO STRING
VAR_INPUT
	WINDEX : WORD;
END_VAR
END_METHOD

METHOD GETBASETYPE_INTERNAL : REFERENCE TO TypeDesc
END_METHOD

METHOD GETENUMMEMBERATTRIBUTELIST_INTERNAL : POINTER TO EnumAttributes
VAR_INPUT
	PNNUMOFENUMVALUES : POINTER TO INT;
	PRESULT : POINTER TO RTS_IEC_RESULT;
END_VAR
END_METHOD

METHOD GETENUMVALUES_INTERNAL : POINTER TO EnumValues
VAR_INPUT
	PNNUMOFENUMVALUES : POINTER TO INT;
	PRESULT : POINTER TO RTS_IEC_RESULT;
END_VAR
END_METHOD

METHOD GETNAME_INTERNAL : POINTER TO STRING
VAR_INPUT
	PRESULT : POINTER TO SysTypes.RTS_IEC_RESULT;
END_VAR
END_METHOD

METHOD GETNATIVESIZE2_INTERNAL : __XWORD
VAR_INPUT
	VARINFO : REFERENCE TO VariableInformation;
END_VAR
END_METHOD

METHOD GETNATIVESIZE_INTERNAL : __XWORD
END_METHOD

METHOD GETNUMOFATTRIBUTES_INTERNAL : WORD
END_METHOD

METHOD GETRANGE_INTERNAL : BOOL
VAR_INPUT
	PLOWER : POINTER TO LWORD;
	PUPPER : POINTER TO LWORD;
END_VAR
END_METHOD

METHOD GETREFERENCEBASETYPE_INTERNAL : REFERENCE TO TypeDesc
VAR_INPUT
	PRESULT : POINTER TO RTS_IEC_RESULT;
END_VAR
END_METHOD

METHOD GETSIZE2_INTERNAL : __XWORD
VAR_INPUT
	VARINFO : REFERENCE TO VariableInformation;
END_VAR
END_METHOD

METHOD GETSIZE_INTERNAL : __XWORD
END_METHOD

METHOD GETSWAPSIZE_INTERNAL : __XWORD
END_METHOD

METHOD GETTYPECLASS2_INTERNAL : TypeClass
VAR_INPUT
	DWFLAGS : DWORD;
END_VAR
END_METHOD

METHOD GETTYPECLASS_INTERNAL : TypeClass
END_METHOD

METHOD GETTYPEDESCVARLENARRAY_INTERNAL : RTS_IEC_RESULT
VAR_INPUT
	PTYPEDESCSTRUCT : POINTER TO TypeDescVarArrayAsStruct;
END_VAR
END_METHOD

METHOD GETTYPEDESC_INTERNAL : UDINT
VAR_INPUT
	PTYPEDESCSTRUCT : POINTER TO TypeDescAsUnion;
END_VAR
END_METHOD

METHOD GETTYPENODE_INTERNAL : REFERENCE TO TypeDesc
VAR_INPUT
	VARINFO : REFERENCE TO VariableInformation;
	OPTIONS : WORD;
END_VAR
END_METHOD

METHOD GETUABUILTINTYPE_INTERNAL : OpcUa_BuiltInType
END_METHOD

METHOD SWAP_INTERNAL : __XWORD
VAR_INPUT
	PDATA : POINTER TO BYTE;
	VARINFO : REFERENCE TO VariableInformation;
	DWSIZE : __XWORD;
	BMOTOROLA : BOOL;
	PRESULT : POINTER TO UDINT;
END_VAR
END_METHOD

METHOD PROTTOKENLENGTH : DINT
VAR_INPUT
	PST : POINTER TO STRING;
END_VAR
END_METHOD

(* ---- TYPEDESC_VARLENARRAY.pou ---- *)
FUNCTION_BLOCK TYPEDESC_VARLENARRAY EXTENDS TypeDesc
VAR
	_IDIMENSIONS : USINT;
	_DIMINFOOFFSET : __XWORD;
	_IDIMINFOTYPEDESC : REFERENCE TO TypeDesc;
	_IBASETYPEDESC : REFERENCE TO TypeDesc;
END_VAR
END_FUNCTION_BLOCK

METHOD FINDCHILD : ITreeWalker
VAR_INPUT
	PSTPATH : POINTER TO STRING;
	VARINFO : REFERENCE TO VariableInformation;
	PRESULT : POINTER TO UDINT;
END_VAR
VAR_IN_OUT
	IOFFSETINPATH : __XWORD;
END_VAR
END_METHOD

METHOD GETNATIVESIZE2_INTERNAL : __XWORD
VAR_INPUT
	VARINFO : REFERENCE TO VariableInformation;
END_VAR
END_METHOD

METHOD GETNATIVESIZE_INTERNAL : __XWORD
END_METHOD

METHOD GETSIZE2_INTERNAL : __XWORD
VAR_INPUT
	VARINFO : REFERENCE TO VariableInformation;
END_VAR
END_METHOD

METHOD GETSIZE_INTERNAL : __XWORD
END_METHOD

METHOD GETTYPECLASS2_INTERNAL : TypeClass
VAR_INPUT
	DWFLAGS : DWORD;
END_VAR
END_METHOD

METHOD GETTYPECLASS_INTERNAL : TypeClass
END_METHOD

METHOD GETTYPEDESCVARLENARRAY_INTERNAL : RTS_IEC_RESULT
VAR_INPUT
	PTYPEDESCSTRUCT : POINTER TO TypeDescVarArrayAsStruct;
END_VAR
END_METHOD

METHOD GETTYPEDESC_INTERNAL : UDINT
VAR_INPUT
	PTYPEDESCSTRUCT : POINTER TO TypeDescAsUnion;
END_VAR
END_METHOD

METHOD GETTYPENODE_INTERNAL : REFERENCE TO TypeDesc
VAR_INPUT
	VARINFO : REFERENCE TO VariableInformation;
	OPTIONS : WORD;
END_VAR
END_METHOD

METHOD GET_INTERNAL : __XWORD
VAR_INPUT
	PDEST : POINTER TO BYTE;
	PSRC : POINTER TO BYTE;
	VARINFO : REFERENCE TO VariableInformation;
	DWSIZE : __XWORD;
	PRESULT : POINTER TO UDINT;
END_VAR
END_METHOD

METHOD NODEFOUND_INTERNAL : UDINT
VAR_INPUT
	VARINFO : REFERENCE TO VariableInformation;
	BDIRECTCHILDFOUND : BOOL;
END_VAR
END_METHOD

METHOD SET_INTERNAL : __XWORD
VAR_INPUT
	PSRC : POINTER TO BYTE;
	PDEST : POINTER TO BYTE;
	VARINFO : REFERENCE TO VariableInformation;
	DWSIZE : __XWORD;
	PRESULT : POINTER TO UDINT;
END_VAR
END_METHOD

METHOD SWAP_INTERNAL : __XWORD
VAR_INPUT
	PDATA : POINTER TO BYTE;
	VARINFO : REFERENCE TO VariableInformation;
	DWSIZE : __XWORD;
	BMOTOROLA : BOOL;
	PRESULT : POINTER TO UDINT;
END_VAR
END_METHOD
